IF in1 >= in2 AND in1 >= in3 THEN
	max3 := in1;
ELSIF in2 >= in1 AND in2 >= in3 THEN
	max3 := in2;
ELSE
	max3 := in3;
END_IF;

END_FUNCTION

// POUs/String/MESSAGE_4R
FUNCTION_BLOCK MESSAGE_4R
VAR_INPUT
	M0 : STRING(STRING_LENGTH);
	M1 : STRING(STRING_LENGTH);
	M2 : STRING(STRING_LENGTH);
	M3 : STRING(STRING_LENGTH);
	MM : INT := 3;
	ENQ : BOOL := TRUE;
	CLK : BOOL := TRUE;
	T1 : TIME := T#3s;
END_VAR
VAR_OUTPUT
	MX : STRING(STRING_LENGTH);
	MN : INT;
	TR : BOOL;
END_VAR
VAR
	timer : TON;
	edge: BOOL;
END_VAR

(*
version 1.1	27. oct. 2008
programmer 	hugo
tested by	tobias

this function generates a rotation meassage with up to 4 strings.
on each rising edge of EN the next message in line will be displayed.
when EN stays high longer then one cycle, the next message will be displayed automatically after the time T1 is elapsed.
the output MX is the generated message and CX is a counter 0..3 signaling the current message displayed.
the displayed messages are 0 .. MM.

*)

(* check for rising edge on EN *)
TR := FALSE;
IF ENQ THEN
	IF (NOT edge AND clk) OR timer.q THEN
			MN := INC1(MN, MM);
			TR := TRUE;
			timer(in := FALSE);
			CASE MN OF
				0 : MX := M0;
				1 : MX := M1;
				2 : MX := M2;
				3 : MX := M3;
			END_CASE;
	END_IF;
	edge := clk;
	timer( in := CLK, pt := T1);
ELSE
	MX := '';
	MN := 0;
END_IF;




(* revision history
hm	8. oct. 2008	rev 1.0
	original version

hm	27. oct. 2008	rev 1.1
	changed _INC to INC1

*)

END_FUNCTION_BLOCK

// POUs/String/MESSAGE_8
FUNCTION_BLOCK MESSAGE_8
VAR_INPUT
	IN1 : BOOL;
	IN2 : BOOL;
	IN3 : BOOL;
	IN4 : BOOL;
	IN5 : BOOL;
	IN6 : BOOL;
	IN7 : BOOL;
	IN8 : BOOL;
END_VAR
VAR_INPUT CONSTANT
	S1 : STRING(STRING_LENGTH);
	S2 : STRING(STRING_LENGTH);
	S3 : STRING(STRING_LENGTH);
	S4 : STRING(STRING_LENGTH);
	S5 : STRING(STRING_LENGTH);
	S6 : STRING(STRING_LENGTH);
	S7 : STRING(STRING_LENGTH);
	S8 : STRING(STRING_LENGTH);
END_VAR
VAR_OUTPUT
	M : STRING(STRING_LENGTH);
END_VAR
VAR
END_VAR

(*
version 1.1	29. mar. 2008
programmer 	hugo
tested by	tobias

this function generates one out of 4 messages specified by S1 .. S8.
the selected message will be presented at the output M.
In1 has higher priority then In2 which has higher priority then IN3 and in8 has the lowest priority.
*)

(* check if an alarm is present if yes set the output M otherwise clear M *)
IF in1 THEN
	M := S1;
ELSIF in2 THEN
	M := S2;
ELSIF in3 THEN
	M := S3;
ELSIF in4 THEN
	M := S4;
ELSIF in5 THEN
	M := S5;
ELSIF in6 THEN
	M := S6;
ELSIF in7 THEN
	M := S7;
ELSIF in8 THEN
	M := S8;
ELSE
	M := '';
END_IF;

(* revision history
hm	26.12.2007		rev 1.0
	original version

hm	29. mar. 2008	rev 1.1
	changed STRING to STRING(STRING_LENGTH)
*)

END_FUNCTION_BLOCK

// POUs/Engineering/measurements/METER_STAT
FUNCTION_BLOCK METER_STAT
VAR_INPUT
	IN : REAL;
	DI : DATE;
	RST : BOOL;
END_VAR
VAR_OUTPUT RETAIN
	Last_Day : REAL;
	Current_Day : REAL;
	Last_Week : REAL;
	Current_Week : REAL;
	Last_Month : REAL;
	Current_Month : REAL;
	Last_Year : REAL;
	Current_Year : REAL;
END_VAR
VAR RETAIN
	Year_Start : REAL;
	Month_Start : REAL;
	Week_Start : REAL;
	Day_Start : REAL;
	last_run: DATE;
END_VAR

(*
	version 1.1	7. oct. 2008
	programmer 	oscat
	tested BY	oscat

METER_STAT runs statistics of a metered value, it calculates the current week, day, month and year consumption and stores the corresponding last day, week, month and year value.

*)

IF rst THEN
	Last_Day := 0;
	Current_Day := 0;
	Day_start := IN;
	Last_week := 0;
	Current_week := 0;
	Week_start := in;
	Last_month := 0;
	Current_month := 0;
	month_start := in;
	last_year := 0;
	current_year := 0;
	year_start := in;
ELSE
	Current_Day := IN - Day_Start;
	Current_Week := In - Week_Start;
	Current_Month := IN - Month_Start;
	Current_Year := IN - Year_Start;
END_IF;

IF YEAR_OF_DATE(DI) > YEAR_OF_DATE(last_run) THEN
	(* a new year has started *)
	last_year := current_year;
	current_year := 0;
	year_start := in;
	last_month := current_month;
	current_month := 0;
	month_start := in;
	last_day := current_day;
	current_day := 0;
	day_start := in;
ELSIF MONTH_OF_DATE(DI) > MONTH_OF_DATE(last_run) THEN
	(* a new month has started, january is alrerady done by year change *)
	last_month := current_month;
	current_month := 0;
	month_start := in;
	last_day := current_day;
	current_day := 0;
	day_start := in;
ELSIF day_of_year(di) > day_of_year(last_run) THEN
	(* day has chaged, first day of year and first day of month has already been taken care of *)
	last_day := current_day;
	current_day := 0;
	day_start := in;
END_IF;
IF DAY_OF_WEEK(DI) < DAY_OF_WEEK(last_run) THEN
	(* a new week has started *)
	last_week := current_week;
	current_week := 0;
	week_start := in;
END_IF;
last_run := di;

(* revision history
hm	16. sep. 2007	rev 1.0
	original version

hm	7. oct. 2008	rev 1.1
	changed function year_to_year_of_date
	changed function month to month_of_date
	changed function weekday to day_of_week

*)

END_FUNCTION_BLOCK

// POUs/Mathematical/MID3
FUNCTION MID3 : REAL
VAR_INPUT
	in1 : REAL;
	in2 : REAL;
	in3 : REAL;
END_VAR
VAR
END_VAR

(*
version 1.1	1 jan 2007
programmer 	hugo
tested by		tobias

returns the mid value of 3 real inputs.

*)

IF (in1 <= in2) AND (in1 >= in3) OR (in1 >= in2) AND (in1 <= in3) THEN
	mid3 := in1;
ELSIF (in2 <= in1) AND (in2 >= in3) OR (in2 >= in1) AND (in2 <= in3) THEN
	mid3 := in2;
ELSE
	mid3 := in3;
END_IF;

(*
hm	1.1.2007	rev 1.1
	rewrote the function for better performance

*)

END_FUNCTION

// POUs/Mathematical/MIN3
FUNCTION MIN3 : REAL
VAR_INPUT
	in1 : REAL;
	in2 : REAL;
	in3 : REAL;
END_VAR
VAR
END_VAR

(*
version 1.0	1 jan 2007
programmer 	hugo
tested by		tobias

this function returns the lowest of 3 real values

*)

IF in1 <= in2 AND in1 <= in3 THEN
	min3 := in1;
ELSIF in2 <= in1 AND in2 <= in3 THEN
	min3 := in2;
ELSE
	min3 := in3;
END_IF;

END_FUNCTION

// POUs/Time&Date/MINUTE_OF_DT
FUNCTION MINUTE_OF_DT : INT
VAR_INPUT
	XDT : DT;
END_VAR
VAR
END_VAR


(*
	version 1.0	6. jun. 2008
	programmer 	oscat
	tested BY	oscat

MINUTE_OF_DT returns the current minute (minute of the hour) of a DT variable

*)

MINUTE_OF_DT := DWORD_TO_INT(DT_TO_DWORD(XDT) MOD 3600)/60;


(* revision history
hm		6.9.2008	rev 1.0
	original version


*)

END_FUNCTION

// POUs/Time&Date/MINUTE_TO_TIME
FUNCTION MINUTE_TO_TIME : TIME
VAR_INPUT
	IN : REAL;
END_VAR
VAR
END_VAR

(*
version 1.2	24. feb. 2009
programmer 	hugo
tested by		oscat

converts an amount of minutes in real to time

*)

MINUTE_TO_TIME := DWORD_TO_TIME(REAL_TO_DWORD(IN * 60000.0));


(* revision history
hm	4. aug 2006	rev 1.0
	original version

hm	14. mar 2008	rev 1.1
	rounded the input after the last digit

hm	24. feb. 2009	rev 1.2
	changed input to IN

*)

END_FUNCTION

// POUs/String/MIRROR
FUNCTION MIRROR : STRING(STRING_LENGTH)
VAR_INPUT
	str : STRING(STRING_LENGTH);
END_VAR
VAR
	pi : POINTER TO ARRAY[1..255] OF BYTE;
	po : POINTER TO BYTE;
	lx: INT;
	i: INT;
END_VAR

(*
version 1.1	29. mar. 2008
programmer 	hugo
tested by	tobias

this function reverses an input string.

*)

pi := ADR(str);
po := ADR(mirror);
lx := LEN(str);
FOR i := lx TO 1 BY - 1 DO
	po^ := pi^[i];
	po := po + 1;
END_FOR;
(* close output string *)
po^:= 0;


(* revision histroy
hm	4. feb. 2008	rev 1.0
	original release

hm	29. mar. 2008	rev 1.1
	changed STRING to STRING(STRING_LENGTH)
*)

END_FUNCTION

// POUs/Engineering/signal processing/MIX
FUNCTION MIX : REAL
VAR_INPUT
	A, B : REAL;
	M : REAL;
END_VAR
VAR
END_VAR

(*
version 1.0	19 nov 2007
programmer 	hugo
tested by		tobias

MIX is an analog Mixer. The Output is (1-M)*A + M*B.

*)

MIX := (1-M)*A + M*B;

(* revision history
hm	19. Nov 2007		rev 1.0
	original version
*)

END_FUNCTION

// POUs/Time&Date/MONTH_BEGIN
FUNCTION MONTH_BEGIN : DATE
VAR_INPUT
	idate : DATE;
END_VAR
VAR
END_VAR

(*
version 1.0	15. jun. 2008
programmer 	hugo
tested by	oscat

returns the date for the first day of the current month in the current year.

*)

MONTH_BEGIN := DWORD_TO_DATE(DATE_TO_DWORD(idate) - INT_TO_DWORD(DAY_OF_MONTH(idate) - 1) * 86400);



(* revision history
hm	15. jun. 2008	rev 1.0
	original version	


*)

END_FUNCTION

// POUs/Time&Date/MONTH_END
FUNCTION MONTH_END : DATE
VAR_INPUT
	IDATE : DATE;
END_VAR
VAR
END_VAR

(*
version 1.1	7. oct. 2008
programmer 	hugo
tested by	oscat

returns the date for the last day of the current month in the current year.

*)

MONTH_END := DWORD_TO_DATE(DATE_TO_DWORD(SET_DATE(YEAR_OF_DATE(idate),MONTH_OF_DATE(idate)+1,1)) - 86400);



(* revision history
hm	15. jun. 2008	rev 1.0
	original version	

hm	7. oct. 2008	rev 1.1
	changed function year to year_of_date
	changed function month to month_of_date

*)

END_FUNCTION

// POUs/Engineering/conversion/MS_TO_BFT
FUNCTION MS_TO_BFT : INT
VAR_INPUT
	MS : REAL;
END_VAR
VAR
END_VAR

(*
version 1.0	12. jun 2008
programmer 	hugo
tested by	oscdat

this function converts wind speed from M/s to beaufort
*)

MS_TO_BFT := REAL_TO_INT(EXPT(MS * 1.196172, 0.666667));


(* revision history
hm	12. 6. 2008		rev 1.0
	original version

*)

END_FUNCTION

// POUs/Engineering/conversion/MS_TO_KMH
FUNCTION MS_TO_KMH : REAL
VAR_INPUT
	ms : REAL;
END_VAR
VAR
END_VAR

(*
version 1.0	4 Feb 2007
programmer 	hugo
tested by		tobias

this function converts velocities from Meters / Second to Kilometers / hour.

*)

MS_TO_KMH := ms * 3.6;

END_FUNCTION

// POUs/Mathematical/MUL_ADD
FUNCTION MUL_ADD : REAL
VAR_INPUT
	X : REAL;
	K : REAL;
	O : REAL;
END_VAR
VAR
END_VAR

(*
version 1.1	11 nov 2007
programmer 	hugo
tested by		tobias

this function multiplies an input X with K and adds Offset O to the result.

*)

MUL_ADD := X * K + O;

(* revision history
hm	28. feb 2007
	original version

hm	11.nov 2007		rev 1.1
	deleted preset values for K and O this makes no sense for a function

*)

END_FUNCTION

// POUs/Engineering/sensor/MULTI_IN
FUNCTION MULTI_IN : REAL
VAR_INPUT
	in_1 : REAL;
	in_2 : REAL;
	in_3 : REAL;
	default : REAL;
	in_min : REAL;
	in_max : REAL;
	mode : BYTE;
END_VAR
VAR
	count: INT;
	F1: BOOL;
	F2: BOOL;
	F3: BOOL;
END_VAR

(*

version 1.2	14. oct. 2008
programmer 	oscat
tested by	oscat

multi_in is a signal conditioning function which can be configured in 8 different ways.
it is used to read multiple sensors for the same value and protect the user from broken sensors or invalid data from sensors.

multi_in can be configured in different ways:
	mode = 0 means the the avg of the 3 inputs is used, this mode is the default mode.
	mode = 1 means in_1 is used.
	mode = 2 means in_2 is used.
	mode = 3 means in_3 is used.
	mode = 4 means default is used.
	mode = 5 means the lowest of the 3 external temperatures is used.
	mode = 6 means the higest externnal temperature is used.
	mode = 7 means the midlle input is used, if there are only two working, the lowest input is used.
	mode > 7 ,eans output is 0 at all times.
	in any config mode, an input higher then in_max or lower then in_min is ignored to prevent values from broken sensors or wires.
	if all inputs are higher then in_max or lower then in_min, a default value (default) is used.
*)

F1 :=  in_1 > in_min AND in_1 < in_max;
F2 :=  in_2 > in_min AND in_2 < in_max;
F3 :=  in_3 > in_min AND in_3 < in_max;

CASE mode OF
0:	count := 0;
	IF F1 THEN
		count := count + 1;
		MULTI_IN := in_1;
	ELSE
		MULTI_IN := 0;
	END_IF;
	IF F2 THEN
		count := count + 1;
		MULTI_IN := MULTI_IN + in_2;
	END_IF;
	IF F3 THEN
		count := count + 1;
		MULTI_IN := MULTI_IN + in_3;
	END_IF;
	IF count = 0 THEN
		MULTI_IN := default;
	ELSE
		MULTI_IN := MULTI_IN / count;
	END_IF;

1:	IF F1 THEN MULTI_IN := in_1; ELSE MULTI_IN := default; END_IF;

2:	IF F2 THEN MULTI_IN := in_2; ELSE MULTI_IN := default; END_IF;

3:	IF F3 THEN MULTI_IN := in_3; ELSE MULTI_IN := default; END_IF;

4:	MULTI_IN := default;

5:	IF F1 THEN MULTI_IN := in_1; ELSE MULTI_IN := in_max; END_IF;
	IF F2 AND in_2 < MULTI_IN THEN MULTI_IN := in_2; END_IF;
	IF F3 AND in_3 < MULTI_IN THEN MULTI_IN := in_3; END_IF;
	IF MULTI_IN = in_max THEN MULTI_IN := default; END_IF;

6:	IF F1 THEN MULTI_IN := in_1; ELSE MULTI_IN := in_min; END_IF;
	IF F2 AND in_2 > MULTI_IN THEN MULTI_IN := in_2; END_IF;
	IF F3 AND in_3 > MULTI_IN THEN MULTI_IN := in_3; END_IF;
	IF MULTI_IN = in_min THEN MULTI_IN := default; END_IF;

7:	IF F1 AND F2 AND F3 THEN MULTI_IN := MID3(in_1, in_2, in_3);
	ELSIF F1 AND F2 THEN MULTI_IN := MIN(in_1, in_2);
	ELSIF F1 AND F3 THEN MULTI_IN := MIN(in_1, in_3);
	ELSIF F2 AND F3 THEN MULTI_IN := MIN(in_2, in_3);
	ELSIF F1 THEN MULTI_IN := in_1;
	ELSIF F2 THEN MULTI_IN := in_2;
	ELSIF F3 THEN MULTI_IN := in_3;
	ELSE MULTI_IN := default;
	END_IF;

END_CASE;

(*
hm 1.1.2007			rev 1.1
	changed midr to mid3 function

hm	14. 10. 2008	rev 1.2
	corrected an error for in_3 overrange detection
	improved performance


*)

END_FUNCTION

// POUs/Logic/gate logic/MUX_2
FUNCTION MUX_2 : BOOL
VAR_INPUT
	D0: BOOL;
	D1: BOOL;
	A0: BOOL;
END_VAR
VAR
END_VAR

(*
	version 1.2	16. oct. 2008
	programmer 	hugo
	tested BY	oscat

	dual input multiplexer
	depending on the value of A0, D0 or D1 will be switched to the Output

	executioin TIME on wago 750-841 = 7us
*)

MUX_2 := SEL(A0, D0, D1);


(*
revision history:
hm	5.10.2006		rev 1.1
	changed to ST Langage for better portability.

hm	16. oct. 2008	rev 1.2
	improved performance

*)

END_FUNCTION

// POUs/Logic/gate logic/MUX_4
FUNCTION MUX_4 : BOOL
VAR_INPUT
	D0: BOOL;
	D1: BOOL;
	D2: BOOL;
	D3: BOOL;
	A0: BOOL;
	A1: BOOL;
END_VAR
VAR
END_VAR

(*
version 1.2	16. oct. 2008
programmer 	hugo
tested BY	oscat

quad input multiplexer
depending on the value of A0 and A1, one of the 4 inputs will be switched to the Output


*)

IF A1 THEN
	MUX_4 := SEL(A0, D2, D3);
ELSE
	MUX_4 := SEL(A0, D0, D1);
END_IF;


(*
revision history:
hm 	5.10.2006		rev 1.1
	rewritten to ST for better portability

hm	16. oct. 2008	rev 1.2
	improved performance

*)

END_FUNCTION

// POUs/Engineering/signal processing/MUX_R2
FUNCTION MUX_R2 : REAL
VAR_INPUT
	IN0 : REAL;
	IN1 : REAL;
	A : BOOL;
END_VAR
VAR
END_VAR

(*
version 1.1	16. oct. 2008
programmer 	oscat
tested by	oscat

MUX_R2 is an analog Multiplexer.
one of 2 real inputs are selected and put through to out.
The Adress input A selects between 2 Real inputs IN0 and IN1, A=0 > In0, A=1 > in1.

*)

MUX_R2 := SEL(A, IN0, IN1);


(* revision history
hm	19. jan. 2007	rev 1.0
	original version

hm	16. oct. 2008	rev 1.1
	improved performance


*)

END_FUNCTION

// POUs/Engineering/signal processing/MUX_R4
FUNCTION MUX_R4 : REAL
VAR_INPUT
	IN0 : REAL;
	IN1 : REAL;
	IN2 : REAL;
	IN3 : REAL;
	A0 : BOOL;
	A1 : BOOL;
END_VAR
VAR
END_VAR

(*
version 1.1	16. oct. 2008
programmer 	oscat
tested by	oscat

MUX_R4 is an analog Multiplexer.
one of 4 real inputs are selected and put through to out.
The Adress input A0 and A1 selects between the 4 Real inputs IN0.. IN1.

*)

IF A1 THEN
	MUX_R4 := SEL(A0, IN2, IN3);
ELSE
	MUX_R4 := SEL(A0, IN0, IN1);
END_IF;



(* revision history
hm	19. jan 2007	rev 1.0
	original version

hm	16. oct. 2008	rev 1.1
	improved performance
*)

END_FUNCTION

// POUs/Mathematical/NEGX
FUNCTION NEGX : REAL
VAR_INPUT
	X : REAL;
END_VAR
VAR
END_VAR


(*
version 1.0	26. oct. 2008
programmer 	hugo
tested by	tobias

This function returns -X

*)

NEGX := -X;




(* revision history
hm	26. oct. 2008	rev 1.0
	original version


*)

END_FUNCTION

// POUs/Engineering/signal processing/OFFSET2
FUNCTION OFFSET2 : REAL
VAR_INPUT
	X : REAL;
	O1, O2, O3, O4 : BOOL;
	D : BOOL;
END_VAR
VAR_INPUT CONSTANT
	Offset_1 : REAL;
	Offset_2 : REAL;
	Offset_3 : REAL;
	Offset_4 : REAL;
	default : REAL;
END_VAR

(*
version 1.0	12 jan 2007
programmer 	oscat
tested by		tobias

The Function offset adds offsets to an analog signal depending on digital inputs.
one offset can be added at the same time, if more then one input is true, the one with the highest number (o1 .. o4) will be used.
The input D will select a default value instead of X for input.

*)

IF D THEN OFFSET2 := default; ELSE OFFSET2 := X; END_IF;
IF O4 THEN OFFSET2 := OFFSET2 + offset_4;
ELSIF O3 THEN OFFSET2 := OFFSET2 + offset_3;
ELSIF O2 THEN OFFSET2 := OFFSET2 + offset_2;
ELSIF O1 THEN OFFSET2 := OFFSET2 + offset_1;
END_IF;

END_FUNCTION

// POUs/Engineering/conversion/OM_TO_F
FUNCTION OM_TO_F : REAL
VAR_INPUT
	OM : REAL;
END_VAR
VAR
END_VAR

(*
version 1.1	18. oct. 2008
programmer 	hugo
tested by		tobias

this function converts Omega F to frequency
F = OM / (2*PI)
*)

OM_TO_F := OM / math.PI2;


(* revision history
hm	22. jan. 2007	rev 1.0
	original version

hm	18. oct. 2008	rev 1.1
	using math constants

*)

END_FUNCTION

// POUs/Other/OSCAT_VERSION
FUNCTION OSCAT_VERSION : DWORD
VAR_INPUT
	IN : BOOL;
END_VAR
VAR
END_VAR


(*
version 1.1	16 dec 2007
programmer 	hugo
tested by		oscat

oscat_version returns the version number in dword format
132 is library version 1.32
if IN = true, the release date will be returned

*)

IF in THEN
	OSCAT_VERSION := DATE_TO_DWORD(D#2009-3-1);
ELSE
	OSCAT_VERSION := 304;
END_IF;

(* revision history
hm	6. oct 2006	rev 1.0
	original version

hm	16. dec 2007	rev 1.1
	added possibility to return date and version depending on IN.

*)

END_FUNCTION

// POUs/Engineering/automation/PARSET
FUNCTION_BLOCK PARSET
VAR_INPUT
	A0, A1 : BOOL;
END_VAR
VAR_INPUT CONSTANT
	X01, X02, X03, X04 : REAL;
	X11, X12, X13, X14 : REAL;
	X21, X22, X23, X24 : REAL;
	X31, X32, X33, X34 : REAL;
	TC : TIME;
END_VAR
VAR_OUTPUT
	P1, P2, P3, P4 : REAL;
END_VAR
VAR
	X : ARRAY[0..3,1..4] OF REAL;
	S1, S2, S3, S4 : REAL;
	tx, last : DWORD;
	start : BOOL;
	set : BYTE;
	init: BOOL;
END_VAR

(*
version 1.1	16. mar. 2008
programmer 	hugo
tested by		tobias

parset selects on of 4 parameter sets adressed by the inputs A0 and A1. if TC is specified, the change of the outputs
is ramped by the time tc
*)

(* read system_time *)
tx := T_PLC_MS();

(* init sequence *)
IF NOT init THEN
	set.0 := NOT A0;
	init := TRUE;
	X[0,1] := X01;
	X[0,2] := X02;
	X[0,3] := X03;
	X[0,4] := X04;
	X[1,1] := X11;
	X[1,2] := X12;
	X[1,3] := X13;
	X[1,4] := X14;
	X[2,1] := X21;
	X[2,2] := X22;
	X[2,3] := X23;
	X[2,4] := X24;
	X[3,1] := X31;
	X[3,2] := X32;
	X[3,3] := X33;
	X[3,4] := X34;
	P1 := X01;
	P2 := X02;
	P3 := X03;
	P4 := X04;
END_IF;

(* check for input change *)
IF (A0 XOR set.0) OR (A1 XOR set.1) THEN
	(* a new set is selected *)
	set.0 := A0;
	set.1 := A1;
	IF tc > t#0s THEN
		start := TRUE;
		last := tx;
		(* save the step speed for the output changes in S *)
		S1 := (X[set,1] - P1)/DWORD_TO_REAL(TIME_TO_DWORD(tc));
		S2 := (X[set,2] - P2)/DWORD_TO_REAL(TIME_TO_DWORD(tc));
		S3 := (X[set,3] - P3)/DWORD_TO_REAL(TIME_TO_DWORD(tc));
		S4 := (X[set,4] - P4)/DWORD_TO_REAL(TIME_TO_DWORD(tc));
	END_IF;
ELSIF start AND tx - last < TIME_TO_DWORD(tc) THEN
	(* ramp the outputs to the new value *)
	P1 := X[set,1] - S1 * DWORD_TO_REAL(TIME_TO_DWORD(Tc) - tx + last);
	P2 := X[set,2] - S2 * DWORD_TO_REAL(TIME_TO_DWORD(Tc) - tx + last);
	P3 := X[set,3] - S3 * DWORD_TO_REAL(TIME_TO_DWORD(Tc) - tx + last);
	P4 := X[set,4] - S4 * DWORD_TO_REAL(TIME_TO_DWORD(Tc) - tx + last);
ELSE
	(* make sure outputs match the correct set values *)
	start := FALSE;
	P1 := X[set,1];
	P2 := X[set,2];
	P3 := X[set,3];
	P4 := X[set,4];
END_IF;

(* revision history
hm	2.11.2007		rev 1.0
	original version

hm	16. mar. 2008	rev 1.1
	added type conversions to avoid warnings under codesys 3.0

*)

END_FUNCTION_BLOCK

// POUs/Engineering/automation/PARSET2
FUNCTION_BLOCK PARSET2
VAR_INPUT
	X : REAL;
END_VAR
VAR_INPUT CONSTANT
	X01, X02, X03, X04 : REAL;
	X11, X12, X13, X14 : REAL;
	X21, X22, X23, X24 : REAL;
	X31, X32, X33, X34 : REAL;
	L1, L2, L3 : REAL;
	TC : TIME;
END_VAR
VAR_OUTPUT
	P1,P2,P3,P4 : REAL;
END_VAR
VAR
	Pset : parset;
	init: BOOL;
END_VAR

(*
version 1.0	3 nov 2007
programmer 	hugo
tested by	tobias

parset2 selects on of 4 parameter sets depending on the value of X. if TC is specified, the change of the outputs
is ramped by the time TC
*)

(* init sequence *)
IF NOT init THEN
	init := TRUE;
	pset(TC:=TC, X01:=X01, X02:=X02, X03:=X03, X04:=X04, X11:=X11, X12:=X12, X13:=X13, X14:=X14, X21:=X21, X22:=X22, X23:=X23, X24:=X24, X31:=X31, X32:=X32, X33:=X33, X34:=X34);
END_IF;
IF ABS(X) < L1 THEN
	pset(A0 := FALSE, A1 := FALSE);
ELSIF ABS(X) < L2 THEN
	pset(A0 := TRUE, A1 := FALSE);
ELSIF ABS(x) < L3 THEN
	pset(A0 := FALSE, A1 := TRUE);
ELSE
	pset(A0 := TRUE, A1 := TRUE);
END_IF;
P1 := pset.P1;
P2 := pset.P2;
P3 := pset.P3;
P4 := pset.P4;

(* revision history
hm		3.11.2007		rev 1.0
	original version

*)

END_FUNCTION_BLOCK

// POUs/Time&Date/PERIOD2
FUNCTION PERIOD2 : BOOL
VAR_INPUT
	DP : ARRAY[0..3,0..1] OF DATE;
	DX : DATE;
END_VAR
VAR
END_VAR

(*
version 1.0	27. apr. 2008
programmer 	hugo
tested by	tobias

PERIOD2 checks if DX is within one of 4 periods and sets the output true if so.

*)

PERIOD2 := 	(DX >= DP[0,0] AND DX <= DP[0,1]) OR
			(DX >= DP[1,0] AND DX <= DP[1,1]) OR
			(DX >= DP[2,0] AND DX <= DP[2,1]) OR
			(DX >= DP[3,0] AND DX <= DP[3,1]);


(* revision history

hm		27. apr 2008	rev 1.0
	original version


*)

END_FUNCTION

// POUs/Logic/Others/PIN_CODE
FUNCTION_BLOCK PIN_CODE
VAR_INPUT
	CB : BYTE;
	E : BOOL;
END_VAR
VAR_INPUT CONSTANT
	PIN : STRING(8);
END_VAR
VAR_OUTPUT
	TP : BOOL;
END_VAR
VAR
	POS: INT := 1;
END_VAR

(*
version 1.0	30. oct. 2008
programmer 	hugo
tested by	oscat

MATRIX_CODE scans the input of a key_pad (MATRIX) for a sequence of characters.

*)

tp := FALSE;
IF e THEN
	IF CB = CODE(pin, pos) THEN
		pos := pos + 1;
		IF pos > LEN(PIN) THEN
			(* proper code is detected *)
			TP := TRUE;
			pos := 1;
		END_IF;
	ELSE
		pos := 1;
	END_IF;
END_IF;


(* revision history
hm	30. oct. 2008	rev 1.0		
	original version 


*)

END_FUNCTION_BLOCK

// POUs/Mathematical/functions/POLYNOM_INT
FUNCTION POLYNOM_INT : REAL
VAR_INPUT
	X : REAL;
	XY : ARRAY[1..5,0..1] OF REAL;
	Pts : INT;
END_VAR
VAR
	I, J : INT;
	stop: INT;
END_VAR

(*
	version 1.2	22 feb 2008
	programmer 	oscat
	tested BY		oscat

POLYNOM_INT calculates an output based on a Polynom interpolation of up to 5 coordinates given in an array
the indut coordinates have to start at the lowest array position and must be sorted ba ascending X values.

*)

(*make sure n is bound within the array size *)
pts := MIN(pts, 5);

(* this part is only to calculate the polynom parameters, which are then stores in the Y array
	the array values, it is not needed during runtime, unless the parameters will change during runtime
	the remaining code without this setup code can be used within a function to calculate specific functions
	the content of the arrays is then used as constant values within the function *)

FOR i := 1 TO pts DO
	stop := i + 1;
   	FOR j := pts TO stop BY -1 DO
   		XY[j,1] := (XY[j,1] - XY[j-1,1]) / (XY[j,0] - XY[j-i,0]);
	END_FOR;
END_FOR;


(* this part is the actual calculation *)
POLYNOM_INT := 0;
FOR i := pts TO 1 BY -1 DO
       POLYNOM_INT := POLYNOM_INT * (X - XY[i,0]) + XY[i,1];
END_FOR;


(* revision history
hm		8. okt 2007		rev 1.0
	original version

hm		17. dec 2007	rev 1.1
	init makes no sense for a function

hm		22. feb 2008	rev 1.2
	improved performance
*)

END_FUNCTION

// POUs/Engineering/conversion/PT_TO_F
FUNCTION PT_TO_F : REAL
VAR_INPUT
	PT : TIME;
END_VAR
VAR
END_VAR

(*
version 1.0	4 aug 2006
programmer 	hugo
tested by		tobias

this function converts periode time to frequency
*)

PT_to_F := 1000/DWORD_TO_REAL(TIME_TO_DWORD(PT));

END_FUNCTION

// POUs/Building/electrical/PULSE_LENGTH
FUNCTION_BLOCK PULSE_LENGTH
VAR_INPUT
	in : BOOL;
END_VAR
VAR_OUTPUT
	short : BOOL;
	middle : BOOL;
	long : BOOL;
END_VAR
VAR_INPUT CONSTANT
	T_short : TIME := t#100ms;
	T_long : TIME := t#1s;
END_VAR
VAR
	tx : TIME;
	tn: TIME;
	edge : BOOL;
END_VAR

(*
version 1.1	15 sep 2007
programmer 	oscat
tested by	oscat

Pulse_length indicates on 3 outputs if an input pulse had been shorter than T_short (short = True), longer than T_long (long = True) or between T_short and T_long (middle = True).

*)

(* read system time *)
tx := DWORD_TO_TIME(T_PLC_MS());

(* reset outputs, they should only be active 1 cycle *)
short := FALSE;
Middle := FALSE;
long := FALSE;

(* detect rising edge *)
IF in AND NOT edge THEN
	edge := TRUE;
	tn := tx;

(* detect for falling edge *)
ELSIF NOT in AND edge THEN
	edge := FALSE;
	tn := tx - tn;
	IF tn < t_short THEN
		short := TRUE;
	ELSIF tn > t_long THEN
		long := TRUE;
	ELSE
		Middle := TRUE;
	END_IF;

(* generate long pulse as soon as T_long is reached *)
ELSIF in AND tx - tn > t_long THEN
	long := TRUE;
END_IF;


(* revision history

hm	15. feb 2006	rev 1.0
	original version

hm	15 sep 2007		rev 1.1
	replaced Time() with T_PLC_MS for compatibility and performance reasons

*)

END_FUNCTION_BLOCK

// POUs/Building/electrical/PULSE_T
FUNCTION_BLOCK PULSE_T
VAR_INPUT
	IN : BOOL;
	T1 : TIME;
	T2 : TIME;
	RST : BOOL;
END_VAR
VAR_OUTPUT
	Q : BOOL;
END_VAR
VAR
	init: BOOL;
	last: TIME;
	tx: TIME;
	edge: BOOL;
END_VAR


(*
version 1.0	15. jul. 2008
programmer 	hugo
tested by	oscat

PULSE_T generates a pulse of length T2 if the input pulse is shorter than T1.
if the input pulse is longer than T1, the output follows the input.
and rising edge on in will kill a possible output pulse and generate a new pulse instead.

*)

tx := DWORD_TO_TIME(T_PLC_MS());
IF NOT init THEN
	init := TRUE;
	last := tx;
ELSIF RST THEN
	(* asynchronous reset *)
	Q := FALSE;
ELSIF IN AND NOT edge AND NOT Q THEN
	(* a rising edge on in will reversre the output status, if new pulse is startet the start time is stored in last *)
	last := tx;
	Q := TRUE;
ELSIF NOT IN AND edge AND ((tx - last) > T1) THEN
	(* a falling edge on IN will clear the output if in was high for more then T1 *)
	Q := FALSE;
ELSIF (tx - last) >= T2 THEN
	(* timeout for long pulse if second click did not occur or in stays high *)
	Q := FALSE;
END_IF;

edge := IN;

(* revision histroy
hm	15. jul. 2008	rev 1.0
	original release


*)

END_FUNCTION_BLOCK

// POUs/Engineering/signal generators/PWM_PW
FUNCTION_BLOCK PWM_PW
VAR_INPUT
	F : REAL;
	PW : TIME;
END_VAR
VAR_OUTPUT
	Q : BOOL;
END_VAR
VAR
	clk: CLK_PRG;
	pulse: TP_X;
END_VAR

(*
version 1.4	19. oct. 2008
programmer 	oscat
tested BY	oscat

this signal generator generates a square wave signal which is specified by the frequency and the pulse width.
*)

IF F > 0 THEN
	CLK(PT := REAL_TO_TIME(1000/F));
	Pulse(in := clk.Q, pt := pw);
	Q := pulse.Q;
END_IF;

(* revision history

hm	25. feb 2007	rev 1.1
	recoded in st for better performance and better portability

hm	27. nov 2007	rev 1.2
	avoid divide by 0 when F = 0

hm	9. dec 2007		rev 1.3
	corrected an error with F = 0

hm	19. oct. 2008	rev 1.4
	changed type tp_r to TP_x brecause of name change

*)

END_FUNCTION_BLOCK

// POUs/Mathematical/Double Precision/R2_ABS
FUNCTION R2_ABS : REAL2
VAR_INPUT
	X : REAL2;
END_VAR
VAR
END_VAR

(*
version 1.0	21. mar. 2008
programmer 	hugo
tested by		tobias

R2_abs returns the absulute value of a double precision real.

*)

IF X.RX >= 0 THEN
	R2_ABS.RX := X.RX;
	R2_ABS.R1 := X.R1;
ELSE
	R2_ABS.RX := ABS(X.RX);
	R2_ABS.R1 := -X.R1;
END_IF;


(* revision history
hm	21. mar. 2008	rev 1.0
	original version

*)

END_FUNCTION

// POUs/Mathematical/Double Precision/R2_ADD2
FUNCTION R2_ADD2 : REAL2
VAR_INPUT
	X : Real2;
	Y : REAL2;
END_VAR
VAR
END_VAR

(*
version 1.0	20. mar. 2008
programmer 	hugo
tested by		tobias

R2_add2 adds a double precision real to a double precision real which extends the accuracy of a real to twice as many digits

*)

R2_ADD2.R1 := X.R1 + Y.R1;
R2_ADD2.RX := X.RX + Y.RX;


(* revision history
hm		20.3.2008	rev 1.0
	original version

*)

END_FUNCTION

// POUs/Mathematical/Double Precision/R2_MUL
FUNCTION R2_MUL : REAL2
VAR_INPUT
	X : REAL2;
	Y : REAL;
END_VAR
VAR
END_VAR

(*
version 1.0	20. mar. 2008
programmer 	hugo
tested by		tobias

R2_mul multiplies a real with a double real which extends the accuracy of a real to twice as many digits

*)

R2_MUL.RX := X.RX * Y;
R2_MUL.R1 := X.R1 * Y;


(* revision history
hm		20.3.2008	rev 1.0
	original version

*)

END_FUNCTION

// POUs/Engineering/signal processing/RANGE_TO_BYTE
FUNCTION RANGE_TO_BYTE : BYTE
VAR_INPUT
	X : REAL;
	low : REAL;
	high : REAL;
END_VAR
VAR
END_VAR

(*
version 1.0	9. jan 2008
programmer 	hugo
tested by		tobias

Range_to_byte converts a real value between low and high into a byte

*)

Range_to_Byte := INT_TO_BYTE(TRUNC_INT((LIMIT(low,X,high)-low) * 255.0 / (high - low)));


(* revision history
hm	9. jan 2008		rev 1.0
	original version

*)

END_FUNCTION

// POUs/Engineering/signal processing/RANGE_TO_WORD
FUNCTION RANGE_TO_WORD : WORD
VAR_INPUT
	X : REAL;
	low : REAL;
	high : REAL;
END_VAR
VAR
END_VAR

(*
version 1.0	9. jan 2008
programmer 	hugo
tested by		tobias

Range_to_word converts a real value between low and high into a byte

*)

Range_to_Word := DINT_TO_WORD(TRUNC_INT((LIMIT(low,X,high)-low) * 65535.0 / (high - low)));


(* revision history
hm	9. jan 2008		rev 1.0
	original version

*)

END_FUNCTION

// POUs/Mathematical/RDMDW
FUNCTION RDMDW : DWORD
VAR_INPUT
	last : DWORD;
END_VAR
VAR
	RX: REAL;
	M: REAL;
END_VAR




(*
version 1.2	18. oct. 2008
programmer 	hugo
tested by		tobias

this function calculates a DWORD pseudo random number.

*)

M := BIT_COUNT(last);
RX := RDM(FRACT(M * math.PI));
RDMDW := SHL(REAL_TO_DWORD(rx*65535),16);
RX := RDM(FRACT(M * math.E));
RDMDW := RDMDW OR (REAL_TO_DWORD(rx*65535) AND 16#0000FFFF);



(* revision history
hm		14. mar 2008		rev 1.0
	original version

hm		18. may. 2008		rev 1.1
	changed constant E to E1

hm		18. oct. 2008		rev 1.2
	using math constants

*)

END_FUNCTION

// POUs/String/REAL_TO_STRF
FUNCTION REAL_TO_STRF : STRING(20)
VAR_INPUT
	IN : REAL;
	N : INT;
END_VAR
VAR
	O: REAL;
	i: INT;
END_VAR

(*
version 1.7	27. feb. 2009
programmer 	hugo
tested by		oscat

Real_to_strF converts a Real to a fixed length String.
the string will be filles with zeroes to achieve the fixed length after the dot.


*)

(* LIMIT N to 0 .. 7 *)
N := LIMIT(0,N,7);
(* round the input to N digits and convert to string *)
O := ABS(in) * EXP10(N);
REAL_TO_STRF := DINT_TO_STRING(REAL_TO_DINT(O));
(* add zeroes in front to make sure sting is at least 8 digits long *)
FOR i := LEN(REAL_TO_STRF) TO N DO REAL_TO_STRF := CONCAT('0', REAL_TO_STRF); END_FOR;
(* add a dot if n > 0 *)
IF n > 0 THEN REAL_TO_STRF := INSERT(REAL_TO_STRF, '.', LEN(REAL_TO_STRF) - N); END_IF;
(* add a minus sign if in is negative *)
IF in < 0 THEN REAL_TO_STRF := CONCAT('-', REAL_TO_STRF); END_IF;


(* revision history
hm	26 jan 2007	rev 1.0
	original version

hm	20. nov. 2007	rev 1.1
	when N=0 ther will be no dot at the end of the string.

hm	15. dec. 2007	rev 1.2
	changed code for better performance

hm	4. mar. 2008	rev 1.3
	result is now rounded instead of trunc

hm	20. mar. 2008	rev 1.4
	changed trunc to real_to_dint because trunc was generating wrong values on wago 842

hm	29. mar. 2008	rev 1.5
	changed STRING to STRING(20)

hm	4. apr. 2008	rev 1.6
	added variable O to avoid an error uner CoDeSys SP PLCWinNT V2.4

hm	27. feb. 2009	rev 1.7
	added a missing zero for IN < 1

*)

END_FUNCTION

// POUs/Mathematical/ROUND
 FUNCTION ROUND : REAL
VAR_INPUT
	in : REAL;
	N : INT;
END_VAR
VAR
	X: REAL;
END_VAR


(*
version 1.5	25. oct. 2008
programmer 	hugo
tested by	tobias

this function rounds a real down to n digits behind the comma.


*)

x := setup.DECADES[LIMIT(0,n,8)];
ROUND := DINT_TO_REAL(REAL_TO_DINT(in * X)) / X;



(* revision history
hm	1. sep 2006	rev 1.0
	original version

hm	2. dec 2007	rev 1.1
	changed code for better performance

hm	8. jan 2008	rev 1.2
	further improvement in performance

hm 11. mar. 2008	rev 1.3
	corrected an error with negative numbers
	use real_to_dint instead of trunc

hm	16. mar 2008	rev 1.4
	added type conversion to avoid warning under codesys 3.0

hm	25. oct. 2008	rev 1.5
	new code using global constants decades
*)

END_FUNCTION

// POUs/String/REPLACE_ALL
FUNCTION REPLACE_ALL : STRING(STRING_LENGTH)
VAR_INPUT
	str : STRING(STRING_LENGTH);
	src : STRING(STRING_LENGTH);
	rep : STRING(STRING_LENGTH);
END_VAR
VAR
	pos: INT;
	lp : INT;
	lx : INT;
END_VAR

(*
version 1.1	29. mar. 2008
programmer 	hugo
tested by	tobias

the function replace_all replaces all occurences of src in str and replaces them by rep.

*)

REPLACE_ALL := str;
lx := LEN(src);
lp := LEN(rep);
pos := FINDP(REPLACE_ALL, src, 1);
WHILE pos > 0 DO
	REPLACE_ALL := REPLACE(REPLACE_ALL,rep,lx, pos);
	pos := FINDP(REPLACE_ALL, src, pos + lp);
END_WHILE;

(* revision histroy
hm	4. feb. 2008	rev 1.0
	original release

hm	29. mar. 2008	rev 1.1
	changed STRING to STRING(STRING_LENGTH)
*)

END_FUNCTION

// POUs/String/REPLACE_CHARS
FUNCTION REPLACE_CHARS : STRING(STRING_LENGTH)
VAR_INPUT
	STR : STRING(STRING_LENGTH);
	SRC : STRING;
	REP : STRING;
END_VAR
VAR
	a, b : INT;
	c: STRING(1);
	stp: INT;
END_VAR

(*
version 1.0		14. may. 2008
programmer 		hugo
tested by			hugo

REPLACE_CHARS erstezt alle character die im string src aufgeführt sind mit dem an der selben stelle im string rep gelisteten character.

*)

REPLACE_CHARS := STR;
(* make sure rep and src are of same length and length is > 0 *)
a := LEN(src);
b := LEN(rep);
IF a < b THEN
	rep := LEFT(rep, a);
ELSIF b < a THEN
	src := LEFT(src, b);
END_IF;

(* search the string and replace if necessary *)
stp := LEN(str);
FOR a := 1 TO stp DO
	c := MID(REPLACE_CHARS, 1, a);
	b := FIND(src, c);
	IF b > 0 THEN
		REPLACE_CHARS := REPLACE(REPLACE_CHARS, MID(rep, 1, b), 1, a);
	END_IF;
END_FOR;



(* revision history
hm	14. may. 2008	rev 1.0
	original version

*)

END_FUNCTION

// POUs/String/REPLACE_UML
FUNCTION REPLACE_UML : STRING(STRING_LENGTH)
VAR_INPUT
	str : STRING(STRING_LENGTH);
END_VAR
VAR
	L : INT;
	pt : POINTER TO BYTE;
	pto : POINTER TO BYTE;
	ptm : POINTER TO BYTE;
	pt1, pt2 : POINTER TO BYTE;
	su : STRING(2);
	pos : INT;
END_VAR

(*
version 1.1	29. mar. 2008
programmer 		kurt
tested by		hugo

REPLACE_UML replaces all occurences of Ä,Ö,Ü and ä,ö,ü,ß with Ae, ae, Oe, oe, Ue, ue and ss.

*)

PT := ADR(str);
pto := ADR(REPLACE_UML);
ptm := pto + INT_TO_DWORD(string_length);
pt1 := ADR(su);
pt2 := pt1 + 1;
L := LEN(str);
WHILE pos < L AND pos < string_length DO
	IF pt^ < 127 THEN
		(* no uml character simlply copy the character*)
		pto^ := pt^;
	ELSE
		(* convert the uml character *)
		su := TO_UML(pt^);
		(* we must make sure pointer are not out of range *)
		pto^ := pt1^;
		IF pto < ptm AND pt2^ > 0 THEN
			pto := pto + 1;
			pto^ := pt2^;
		END_IF;
	END_IF;
	(* increment pointers *)
	pt := pt + 1;
	pto := pto + 1;
	pos := pos + 1;
END_WHILE;

(* properly close the output string *)
pto^ := 0;


(* revision history
hm	29. feb 2008	rev 1.0
	original version

hm	29. mar. 2008	rev 1.1
	changed STRING to STRING(STRING_LENGTH)
	new code to avoid pointer out of range
	use new function to_uml
*)

END_FUNCTION

// POUs/String/TO_UML
FUNCTION TO_UML : STRING(2)
VAR_INPUT
	IN : BYTE;
END_VAR
VAR
END_VAR

(*
version 1.1	17. dec. 2008
programmer 		hugo
tested by		tobias

to_uml converts a character above 127 to a two digit character below 127.
the character Ä is converted to Ae

*)

CASE in OF
	196:	(* Ä *)
		TO_UML := 'Ae';
	214:	(* Ö *)
		TO_UML := 'Oe';
	220:	(* Ü *)
		TO_UML := 'Ue';
	223:	(* ß *)
		TO_UML := 'ss';
	228:	(* ä *)
		TO_UML := 'ae';
	246:	(* ö *)
		TO_UML := 'oe';
	252:	(* ü *)
		TO_UML := 'ue';
ELSE
	TO_UML := CHR_TO_STRING(IN);
END_CASE;



(* revision history
hm	29. mar. 2008	rev 1.0
	original version

hm	17. dec. 2008	rev 1.1
	changes name of function chr to chr_to_string

*)

END_FUNCTION

// POUs/Engineering/sensor/RES_NI
FUNCTION RES_NI : REAL
VAR_INPUT
	T : REAL;
	R0 : REAL;
END_VAR
VAR CONSTANT
	A : REAL := 0.5485;
	B : REAL := 0.665E-3;
	C : REAL := 2.805E-9;
END_VAR
VAR
	T2: REAL;
END_VAR

(*
version 1.2	2 dec 2007
programmer 	hugo
tested by		tobias

this function returs the resistance for a nickel sensor for a temperature range from -60..+180 °C *)

T2 := T*T;
Res_NI := R0 + A*T + B*T2 + C*T2*T2;

(* revision history

hm	4.8.2006		rev 1.0
	original version

hm	13.9.2007		rev 1.1
	changed coding for better performance

hm	2. dec. 2007	rev 1.2
	changed code for better performance
*)

(*

 Auszug aus DIN 43760 für Ni100

°C		R		°C		R		°C	R		°C		R		°C		R

-60 	69,5 	-10 	94,6 	40 	123,0 	90 		154,9 	140 	190,9
-55 	71,9 	-5 		97,3 	45 	126,0 	95 		158,3 	145 	194,8
-50 	74,3 	0 		100,0 	50 	129,1 	100 	161,8 	150 	198,7
-45 	76,7 	5 		102,8 	55 	132,2 	105 	165,3 	155 	202,6
-40 	79,1 	10 		105,6 	60 	135,3 	110 	168,8 	160 	206,6
-35 	81,6 	15 		108,4 	65 	138,5 	115 	172,4 	165 	210,7
-30 	84,2 	20 		111,2 	70 	141,7 	120 	176,0 	170 	214,8
-25 	86,7 	25 		114,1 	75 	145,0 	125 	179,6 	175 	219,0
-20 	89,3 	30 		117,1 	80 	148,3 	130 	183,3 	180 	223,2
-15 	91,9 	35 		120,0 	85 	151,6 	135 	187,1 	  	 

*)

END_FUNCTION

// POUs/Engineering/sensor/RES_NTC
FUNCTION RES_NTC : REAL
VAR_INPUT
	T : REAL;
	RN : REAL;
	B : REAL;
END_VAR


(*
version 1.0	30. dec. 2008
programmer 	hugo
tested by		tobias

this function returs the resistance for a NTC sensor for a given temperature in °C.
RN is the resistance at 25 °C and B is a constant for the given sensor.

*)

RES_NTC := RN * EXP(B * (1/(T+273.15) - 0.00335401643468053));



(* revision history

hm 30. dec. 2008	rev 1.0
	original version


*)

END_FUNCTION

// POUs/Engineering/sensor/RES_PT
FUNCTION RES_PT : REAL
VAR_INPUT
	T : REAL;
	R0 : REAL;
END_VAR
VAR CONSTANT
	A : REAL := 3.90802E-3 ;
	B : REAL := -5.802E-7;
	C : REAL := -4.27350E-12;
END_VAR
VAR
	T2: REAL;
END_VAR

(*
version 1.2	2. dec. 2007
programmer 	hugo
tested by	oscat


this function returs the resistance for a platinum sensor for a temperature range from -200..+850 °C *)

T2 := T * T;

IF T >= 0 THEN
	RES_PT := R0 * ( 1 + A*T + B*T2);
ELSE
	RES_PT := R0 * ( 1 + A*T + B*T2 + C*(T-100)*T2*T);
END_IF;



(* revision history
hm	4. aug. 2006	rev 1.1
	original version

hm	2. dec 2007		rev 1.2
	changed code for better performance


*)


(*
 Auszug aus DIN 43760 für Pt100

°C		R		°C		R		°C	R			°C		R			°C		R			°C		R

-200 	18,49 	-100 	60,25 	0 	100,00 	100 	138,50 	200 	175,84 	300 	212,02
-195 	20,65 	-95 	62,28 	5 	101,95 	105 	140,39 	205 	177,68 	305 	213,80
-190 	22,80 	-90 	64,30 	10 	103,90 	110 	142,29 	210 	179,51 	310 	215,57
-185 	24,94 	-85 	66,31 	15 	105,85 	115 	144,17 	215 	181,34 	315 	217,35
-180 	27,08 	-80 	68,33 	20 	107,79 	120 	146,06 	220 	183,17 	320 	219,12
-175 	29,20 	-75 	70,33 	25 	109,73 	125 	147,94 	225 	184,99 	325 	220,88
-170 	31,32 	-70 	72,33 	30 	111,67 	130 	149,82 	230 	186,82 	330 	222,65
-165 	33,43 	-65 	74,33 	35 	113,61 	135 	151,70 	235 	188,63 	335 	224,41
-160 	35,33 	-60 	76,33 	40 	115,54 	140 	153,58 	240 	190,45 	340 	226,17
-155 	37,63 	-55 	78,32 	45 	117,47 	145 	155,45 	245 	192,26 	345 	227,92
-150 	39,71 	-50 	80,31 	50 	119,40 	150 	157,31 	250 	194,07 	350 	229,67
-145 	41,79 	-45 	82,29 	55 	121,32 	155 	159,18 	255 	195,88 	355 	231,42
-140 	43,87 	-40 	84,27 	60 	123,24 	160 	161,04 	260 	197,69 	360 	233,17
-135 	45,94 	-35 	86,25 	65 	125,16 	165 	162,90 	265 	199,49 	365 	234,91
-130 	48,00 	-30 	88,22 	70 	127,07 	170 	164,76 	270 	201,29 	370 	236,65
-125 	50,06 	-25 	90,19 	75 	128,98 	175 	166,61 	275 	203,08 	375 	238,39
-120 	52,11 	-20 	92,16 	80 	130,89 	180 	168,46 	280 	204,88 	380 	240,13
-115 	54,15 	-15 	94,12 	85 	132,80 	185 	170,31 	285 	206,67 	385 	241,86
-110 	56,19 	-10 	96,09 	90 	134,70 	190 	172,16 	290 	208,45 	390 	243,59
-105 	58,22 	-5 		98,04 	95 	136,60 	195 	174,00 	295 	210,24 	395 	245,31

*)
(*
revision history


*)

END_FUNCTION

// POUs/Engineering/sensor/RES_SI
FUNCTION RES_SI : REAL
VAR_INPUT
	T : REAL;
	RS : REAL;
	TS : REAL;
END_VAR
VAR CONSTANT
	A : REAL := 7.64E-3;
	B : REAL := 1.66E-5;
END_VAR
VAR
	TX: REAL;
END_VAR

(*
version 1.1	2 dec 2007
programmer 	hugo
tested by		tobias

this function returs the resistance for a silicon sensor for a temperature range from -50..+150 °C
for example KTY10 normaly Rs at 25 °C
*)

TX := T - TS;
RES_SI := RS * ( 1 + A * TX + B * TX * TX);

(* revision history
hm		4. aug 2006		rev 1.0
	original version

hm		2. dec 2007		rev 1.1
	changed code for better performance

*)

END_FUNCTION

// POUs/Engineering/signal generators/RMP_SOFT
FUNCTION_BLOCK RMP_SOFT
VAR_INPUT
	IN : BOOL;
	VAL : BYTE;
END_VAR
VAR_INPUT CONSTANT
	PT_ON: TIME;
	PT_OFF : TIME;
END_VAR
VAR_OUTPUT
	OUT : BYTE;
END_VAR
VAR
	rmp : _RMP_B;
	tmp: BYTE;
END_VAR

(*
version 2.0	26. oct. 2008
programmer 	oscat
tested BY		oscat

this soft on/off ramp generator generates a soft on and soft off ramp while the max on value is set by the input
the time for a full ramp can be set by config variables for up and down ramp.

*)

tmp := SEL(in, 0, val);
IF tmp > out THEN
	(* we need to ramp down *)
	rmp(dir := TRUE, E := TRUE, TR := PT_ON, rmp := out);
	(* make sure out does not surpass tmp *)
	out := MIN(out, tmp);
ELSIF tmp < out THEN
	(* we need to ramp up *)
	rmp(dir := FALSE, E := TRUE, TR := PT_OFF, rmp := out);
	(* make sure out does not surpass tmp *)
	out := MAX(out, tmp);
ELSE
	(* no ramp necessary *)
	rmp(E := FALSE, rmp := out);
END_IF;


(* revision history

hm 22.1.2007	rev 1.1
	deleted unused variables X1 and I, X2 and X3

hm	17.9.2007	rev 1.2
	replaced time() with t_plc_ms() for compatibility reasons

hm	26. oct. 2008	2.0
	new code using _rmp_b
*)

END_FUNCTION_BLOCK

// POUs/Mathematical/RND
FUNCTION RND : REAL
VAR_INPUT
	X : REAL;
	N : INT;
END_VAR
VAR
	M : REAL;
END_VAR

(*
version 1.1	26. oct. 2008
programmer 	hugo
tested by	tobias

this function rounds a real down to n digits total.
round(3.1415,2) = 3.1

*)

IF X = 0 THEN
	RND := 0;
ELSE
	M := EXPN(10,N - CEIL(LOG(ABS(X))));
	RND := DINT_TO_REAL(REAL_TO_DINT(X * M)) / M;
END_IF;



(* revision history
hm	11. mar 2008	rev 1.0
	original version

hm	26. oct. 2008	rev 1.1
	code optimization
*)

END_FUNCTION

// POUs/Time&Date/RTC_2
FUNCTION_BLOCK RTC_2
VAR_INPUT
	SET : BOOL;
	SDT : DT;
	SMS : INT;
	DEN : BOOL;
	OFS : INT;
END_VAR
VAR_OUTPUT
	UDT : DT;
	LDT : DT;
	DSO : BOOL;
	XMS : INT;
END_VAR
VAR
	RT : RTC_MS;
END_VAR

(*
version 1.2	12. jun. 2008
programmer 	hugo
tested by	tobias

RTC_2 is a real time clock module which runs utc and generates local time from utc.
daylight savings time can be enabled with den and an additional local time is generated with a delay of ofs.

*)

(* call rtc *)
RT(SET := SET, SDT := SDT, SMS := SMS);
UDT := rt.xdt;
XMS := rt.XMS;

(* check for daylight savings time and set dso output *)
DSO := DST(udt) AND DEN;

(* calculate time offset and set ldt output *)
LDT := DWORD_TO_DT(DT_TO_DWORD(UDT) + INT_TO_DWORD(ofs + BOOL_TO_INT(DSO)) * 3600);


(* revision history
hm		20. jan. 2008	rev 1.0
	original version

hm		20. feb. 2008	rev 1.1
	added Millisecond Set input

hm		12. jun. 2008	rev 1.2
	improved performance
*)

END_FUNCTION_BLOCK

// POUs/Time&Date/RTC_MS
FUNCTION_BLOCK RTC_MS
VAR_INPUT
	SET : BOOL;
	SDT : DT;
	SMS : INT;
END_VAR
VAR_OUTPUT
	XDT : DT;
	XMS : INT;
END_VAR
VAR
	init: BOOL;
	last: DWORD;
	Tx: DWORD;
END_VAR

(*
version 1.1	20. feb. 2008
programmer 	hugo
tested by	tobias

RTC_MS is a real time clock module which can be set to SDT when set is TRUE and the outputs XDT and XT present the DateTime and TOD with a resolution of milliseconds.

*)

tx := T_PLC_MS();
IF set OR NOT init THEN
	(* clock needs to be set when set is true or after power up *)
	init := TRUE;
	xdt := SDT;
	XMS := SMS;
ELSE
	XMS := XMS + DWORD_TO_INT(tx - last);
	(* check if one second has expired *)
	IF XMS > 999 THEN
		XDT := XDT + T#1s;
		XMS := XMS - 1000;
	END_IF;
END_IF;
last := tx;


(* revision history
hm		20. jan. 2008	rev 1.0
	original version

hm		20. feb. 2008	rev 1.1
	added Millisecond Set input
*)

END_FUNCTION_BLOCK

// POUs/Engineering/signal processing/SCALE_B
FUNCTION SCALE_B : REAL
VAR_INPUT
	X : BYTE;
	I_LO : BYTE;
	I_HI : BYTE;
	O_LO : REAL;
	O_HI : REAL;
END_VAR
VAR
END_VAR

(*
version 1.0	18. may. 2008
programmer 	hugo
tested by		tobias

Scale_B is used to translate and scale a byte input x to a real output.

*)

SCALE_B := (O_HI - O_LO) / BYTE_TO_REAL(I_HI - I_LO) * BYTE_TO_REAL(LIMIT(I_LO,X,I_HI));


(* revision history
hm	18. may. 2008		rev 1.0
	original version
*)

END_FUNCTION

// POUs/Engineering/signal processing/SCALE_B2
FUNCTION SCALE_B2 : REAL
VAR_INPUT
	in1: BYTE;
	in2: BYTE;
	K : REAL;
	O : REAL;
END_VAR
VAR_INPUT CONSTANT
	in1_min: REAL;
	in1_max: REAL := 1000;
	in2_min: REAL;
	in2_max: REAL := 1000;
END_VAR

(*
version 1.4	3. nov. 2008
programmer 	hugo
tested by	oscat

this functiob block can scale up to two inputs.
inputs have their min value at 0 and their max value at 255 while the min and max value can be either positive or negative.
inputs ramp between min and max values for the respective inputs to be between (0..255).
the summed output is then scaled by an scale input K and a offset O can be added to the output.
min and max input configurations can be edited in the cfc editor by double clicking the symbol body.

*)

SCALE_B2 := 	(((in1_max - in1_min)* in1 + (in2_max - in2_min)* in2) * 0.003921569 + in1_min + in2_min) * K + O;

(* code bofore rev 1.2
scale_B2 := 	((in1_max - in1_min)* in1 / 255 + in1_min +
				(in2_max - in2_min)* in2 / 255 + in2_min)
				* K + O;
*)

(* revision History
hm 19.1.2007		rev 1.1
	changed outputs to real to avoid overflow of integer
	added offset for better cascading of scale functions
	changed from FB to function

hm	6. jan 2008		rev 1.2
	improved performance

hm	26. oct. 2008	rev 1.3
	code optimization

hm	3. nov. 2008	rev 1.4
	used wrong factor in formula

*)

END_FUNCTION

// POUs/Engineering/signal processing/SCALE_B4
FUNCTION SCALE_B4 : REAL
VAR_INPUT
	in1: BYTE;
	in2: BYTE;
	in3: BYTE;
	in4: BYTE;
	K : REAL;
	O : REAL;
END_VAR
VAR_INPUT CONSTANT
	in1_min: REAL;
	in1_max: REAL := 1000;
	in2_min: REAL;
	in2_max: REAL := 1000;
	in3_min: REAL;
	in3_max: REAL := 1000;
	in4_min: REAL;
	in4_max: REAL := 1000;
END_VAR

(*
version 1.4	3. nov. 2008
programmer 	hugo
tested by	tobias

	this functiob block can scale up to 4 inputs.
	the inputs have their min value at 0 and their max value at 255 while the min and max value can be either positive or negative.
	the inputs ramp between min and max values for the respective inputs to be between (0..255).
	the summed output is then scaled by an scale input K and a offset O can be added to the output.
	the min and max input configurations can be edited in the cfc editor by double clicking the symbol body.

*)

SCALE_B4 := 	(((in1_max - in1_min)* in1 + (in2_max - in2_min)* in2 + (in3_max - in3_min)* in3 + (in4_max - in4_min)* in4)* 0.003921569 + in1_min + in2_min + in3_min + in4_min) * K + O;


(* revision History
hm 19.1.2007		rev 1.1
	changed outputs to real to avoid overflow of integer
	added offset for better cascading of scale functions
	changed from fb to function

hm	6. jan 2008		rev 1.2
	improved performance

hm	26. oct. 2008	rev 1.3
	optimized code

hm	3. nov. 2008	rev 1.4
	used wrong factor in formula

*)

END_FUNCTION

// POUs/Engineering/signal processing/SCALE_B8
FUNCTION SCALE_B8 : REAL
VAR_INPUT
	in1: BYTE;
	in2: BYTE;
	in3: BYTE;
	in4: BYTE;
	in5: BYTE;
	in6: BYTE;
	in7: BYTE;
	in8: BYTE;
	K : REAL;
	O : REAL;
END_VAR
VAR_INPUT CONSTANT
	in1_min: REAL;
	in1_max: REAL := 1000;
	in2_min: REAL;
	in2_max: REAL := 1000;
	in3_min: REAL;
	in3_max: REAL := 1000;
	in4_min: REAL;
	in4_max: REAL := 1000;
	in5_min: REAL;
	in5_max: REAL := 1000;
	in6_min: REAL;
	in6_max: REAL := 1000;
	in7_min: REAL;
	in7_max: REAL := 1000;
	in8_min: REAL;
	in8_max: REAL := 1000;
END_VAR

(*
version 1.4	3. nov. 2008
programmer 	hugo
tested by	oscat

this functiob block can scale up to 8 inputs.
the inputs have their min value at 0 and their max value at 255 while the min and max value can be either positive or negative.
the inputs ramp between min and max values for the respective inputs to be between (0..255).
the summed output is then scaled by an scale input K and a offset O can be added to the output.
the min and max input configurations can be edited in the cfc editor by double clicking the symbol body.

*)

SCALE_B8 := 	(((in1_max - in1_min)* in1 + (in2_max - in2_min)* in2 + (in3_max - in3_min)* in3 + (in4_max - in4_min)* in4 +
				(in5_max - in5_min)* in5 + (in6_max - in6_min)* in6 + (in7_max - in7_min)* in7 + (in8_max - in8_min)* in8) * 0.003921569
				 + in1_min + in2_min + in3_min + in4_min + in5_min + in6_min + in7_min + in8_min) * K + O;


(* revision History
hm	19. jan.2007	rev 1.1
	changed outputs to real to avoid overflow of integer
	added offset for better cascading of scale functions

hm	6. jan. 2008	rev 1.2
	improved performance

hm	26. oct. 2008	rev 1.3
	code optimization

hm	3. nov. 2008	rev 1.4
	used wrong factor in formula

*)

END_FUNCTION

// POUs/Engineering/signal processing/SCALE_D
FUNCTION SCALE_D : REAL
VAR_INPUT
	X : DWORD;
	I_LO : DWORD;
	I_HI : DWORD;
	O_LO : REAL;
	O_HI : REAL;
END_VAR
VAR
END_VAR

(*
version 1.1	13. nov. 2008
programmer 	hugo
tested by	oscat

Scale_D is used to translate and scale a DWORD input x to a real output.
the input is limited to I_LO <= X <= I_HI.

*)

SCALE_D := (O_HI - O_LO) / DWORD_TO_REAL(I_HI - I_LO) * DWORD_TO_REAL(LIMIT(I_LO,X,I_HI) - I_LO) + O_LO;


(* revision history
hm	18. may. 2008	rev 1.0
	original version

hm	13. nov. 2008	rev 1.1
	corrected formula for negative gradient
*)

END_FUNCTION

// POUs/Engineering/signal processing/SCALE_R
FUNCTION SCALE_R : REAL
VAR_INPUT
	X : REAL;
	I_LO : REAL;
	I_HI : REAL;
	O_LO : REAL;
	O_HI : REAL;
END_VAR
VAR
END_VAR

(*
version 1.1	13. nov. 2008
programmer 	hugo
tested by	oscat

Scale_R is used to translate and scale a REAL input x to a real output.
the input is limited to I_LO <= X <= I_HI.

*)

SCALE_R := (O_HI - O_LO) / (I_HI - I_LO) * (LIMIT(I_LO,X,I_HI) - I_LO) + O_LO;


(* revision history
hm	18. may. 2008		rev 1.0
	original version

hm	13. nov. 2008	rev 1.1
	corrected formula for negative gradient

*)

END_FUNCTION

// POUs/Engineering/signal processing/SCALE_X2
FUNCTION SCALE_X2 : REAL
VAR_INPUT
	IN1: BOOL;
	IN2: BOOL;
	K : REAL;
	O : REAL;
END_VAR
VAR_INPUT CONSTANT
	IN1_MIN: REAL;
	IN1_MAX: REAL := 1000;
	IN2_MIN: REAL;
	IN2_MAX: REAL := 1000;
END_VAR

(*
version 1.1	26. oct. 2008
programmer 	hugo
tested by		tobias

	this functiob block can scale up to two inputs.
	the input can select between two values with true or false.
	the summed output is then scaled by an scale input K and a offset O can be added to the output.
	the min and max input configurations can be edited in the cfc editor by double clicking the symbol body.

*)

SCALE_X2 := (SEL(IN1,IN1_MIN, IN1_MAX)+ SEL(IN2,IN2_MIN, IN2_MAX))*k + o;


(* revision history
hm	19. jan, 2007	rev 1.0
	original version

hm	26. oct. 2008	rev 1.1
	code optimized

*)

END_FUNCTION

// POUs/Engineering/signal processing/SCALE_X4
FUNCTION SCALE_X4 : REAL
VAR_INPUT
	IN1: BOOL;
	IN2: BOOL;
	IN3: BOOL;
	IN4: BOOL;
	K : REAL;
	O : REAL;
END_VAR
VAR_INPUT CONSTANT
	IN1_MIN: REAL;
	IN1_MAX: REAL := 1000;
	IN2_MIN: REAL;
	IN2_MAX: REAL := 1000;
	IN3_MIN: REAL;
	IN3_MAX: REAL := 1000;
	IN4_MIN: REAL;
	IN4_MAX: REAL := 1000;
END_VAR

(*
version 1.1	26. oct. 2008
programmer 	hugo
tested by		tobias

	this function can scale up to 4 inputs.
	the input can select between two values with true or false.
	the summed output is then scaled by an scale input K and a offset O can be added to the output.
	the min and max input configurations can be edited in the cfc editor by double clicking the symbol body.

*)

SCALE_X4 := (SEL(IN1,IN1_MIN, IN1_MAX)+ SEL(IN2,IN2_MIN, IN2_MAX)+SEL(IN3,IN3_MIN, IN3_MAX)+ SEL(IN4,IN4_MIN, IN4_MAX))*k + o;


(* revision history
hm	19. jan. 2008	rev 1.0
	original version

hm	26. oct. 2008	rev 1.1
	optimized code
*)

END_FUNCTION

// POUs/Engineering/signal processing/SCALE_X8
FUNCTION SCALE_X8 : REAL
VAR_INPUT
	in1: BOOL;
	in2: BOOL;
	in3: BOOL;
	in4: BOOL;
	in5: BOOL;
	in6: BOOL;
	in7: BOOL;
	in8: BOOL;
	K : REAL;
	O : REAL;
END_VAR
VAR_INPUT CONSTANT
	in1_min: REAL;
	in1_max: REAL := 1000;
	in2_min: REAL;
	in2_max: REAL := 1000;
	in3_min: REAL;
	in3_max: REAL := 1000;
	in4_min: REAL;
	in4_max: REAL := 1000;
	in5_min: REAL;
	in5_max: REAL := 1000;
	in6_min: REAL;
	in6_max: REAL := 1000;
	in7_min: REAL;
	in7_max: REAL := 1000;
	in8_min: REAL;
	in8_max: REAL := 1000;
END_VAR

(*
version 1.2	24. jan. 2009
programmer 	hugo
tested by	oscat

this function can scale up to 4 inputs.
the input can select between two values with true or false.
the summed output is then scaled by an scale input K and a offset O can be added to the output.
the min and max input configurations can be edited in the cfc editor by double clicking the symbol body.

*)

SCALE_X8 := (SEL(IN1,IN1_MIN, IN1_MAX)+ SEL(IN2,IN2_MIN, IN2_MAX)+SEL(IN3,IN3_MIN, IN3_MAX)+ SEL(IN4,IN4_MIN, IN4_MAX)
				+SEL(IN5,IN5_MIN, IN5_MAX)+ SEL(IN6,IN6_MIN, IN6_MAX)+SEL(IN7,IN7_MIN, IN7_MAX)+ SEL(IN8,IN8_MIN, IN8_MAX))*k + o;



(* revision history
hm	19. jan. 2008	rev 1.0
	original version

hm	26. oct. 2008	rev 1.1
	optimized code

hm	24. jan. 2008	rev 1.2
	corrected error in formula
*)

END_FUNCTION

// POUs/Logic/generators/SCHEDULER
FUNCTION_BLOCK SCHEDULER
VAR_INPUT
	E0 : BOOL;
	E1 : BOOL;
	E2 : BOOL;
	E3 : BOOL;
END_VAR
VAR_INPUT CONSTANT
	T0, T1, T2, T3 : TIME;
END_VAR
VAR_OUTPUT
	Q0, Q1, Q2, Q3 : BOOL;
END_VAR
VAR
	init : BOOL;
	s0, s1, s2, s3 : TIME;
	tx : TIME;
	c : INT;
END_VAR


(*
version 1.0	28. sep 2008
programmer 	hugo
tested by		tobias

SCHEDULER is used to call programs or function blocks at specific intervals.
T0..T3 defines the interval times.

*)

(* read system_time *)
tx := DWORD_TO_TIME(T_PLC_MS());

IF NOT init THEN
	init := TRUE;
	s0 := tx - T0;
	s1 := tx - T1;
	s2 := tx - T2;
	s3 := tx - T3;
END_IF;

Q0 := Q1 := Q2 := Q3 :=FALSE;

CASE c OF
	0: 	IF tx - s0 >= T0 THEN
			Q0 := E0;
			s0 := tx;
		END_IF;
		c := 1;
	1: 	IF tx - s1 >= T1 THEN
			Q1 := E1;
			s1 := tx;
		END_IF;
		c := 2;
	2: 	IF tx - s2 >= T2 THEN
			Q2 := E2;
			s2 := tx;
		END_IF;
		c := 3;
	3: 	IF tx - s3 >= T3 THEN
			Q3 := E3;
			s3 := tx;
		END_IF;
		c := 0;
END_CASE;


(* revision history

hm 28. sep. 2008		rev 1.0
	original version


*)

END_FUNCTION_BLOCK

// POUs/Logic/generators/SCHEDULER_2
FUNCTION_BLOCK SCHEDULER_2
VAR_INPUT
	E0 : BOOL;
	E1 : BOOL;
	E2 : BOOL;
	E3 : BOOL;
END_VAR
VAR_INPUT CONSTANT
	C0, C1, C2, C3 : UINT;
	O0, O1, O2, O3 : UINT;
END_VAR
VAR_OUTPUT
	Q0, Q1, Q2, Q3 : BOOL;
END_VAR
VAR
	sx : UINT;
END_VAR


(*
version 1.0	29. sep 2008
programmer 	hugo
tested by		tobias

SCHEDULER_2 is used to call programs or function blocks at specific cycles.
C0..C3 defines after how many cycles the output becomes active.
O0..O3 defines a cycle offset at startup.

*)

Q0 := E0 AND (sx MOD C0 - O0 = 0);
Q1 := E1 AND (sx MOD C1 - O1 = 0);
Q2 := E2 AND (sx MOD C2 - O2 = 0);
Q3 := E3 AND (sx MOD C3 - O3 = 0);

(* increment cycle counter every cycle *)
sx := sx + 1;


(* revision history
hm 29. sep. 2008		rev 1.0
	original version


*)

END_FUNCTION_BLOCK

// POUs/Time&Date/SDT_TO_DATE
FUNCTION SDT_TO_DATE : DATE
VAR_INPUT
	DTI : SDT;
END_VAR
VAR
END_VAR


(*
version 1.0	18. oct 2008
programmer 	hugo
tested by	oscat

converts Structured date time (SDT) to Date Time

*)

SDT_TO_DATE := SET_DATE(DTI.YEAR, DTI.MONTH, DTI.DAY);



(* revision history

hm 18. oct. 2008	rev 1.0
	original version

*)

END_FUNCTION

// POUs/Time&Date/SDT_TO_DT
FUNCTION SDT_TO_DT : DT
VAR_INPUT
	DTI : SDT;
END_VAR
VAR
END_VAR


(*
version 1.0	18. oct 2008
programmer 	hugo
tested by	oscat

converts Structured date time (SDT) to Date Time

*)

SDT_TO_DT := SET_DT(DTI.YEAR, DTI.MONTH, DTI.DAY, DTI.HOUR, DTI.MINUTE, DTI.SECOND);



(* revision history

hm 18. oct. 2008	rev 1.0
	original version

*)

END_FUNCTION

// POUs/Time&Date/SDT_TO_TOD
FUNCTION SDT_TO_TOD : TOD
VAR_INPUT
	DTI : SDT;
END_VAR
VAR
END_VAR


(*
version 1.1	16. nov. 2008
programmer 	hugo
tested by	oscat

converts Structured date time (SDT) to Date Time

*)

SDT_TO_TOD := DWORD_TO_TOD(INT_TO_DWORD(DTI.HOUR) * 3600000 + INT_TO_DWORD(DTI.MINUTE) * 60000 + INT_TO_DWORD(DTI.SECOND) * 1000 + INT_TO_DWORD(DTI.MS));



(* revision history

hm 18. oct. 2008	rev 1.0
	original version

hm	16. nov. 2008	rev 1.1
	added typecasts to avoid warnings
*)

END_FUNCTION

// POUs/Time&Date/SECOND_OF_DT
FUNCTION SECOND_OF_DT : INT
VAR_INPUT
	XDT : DT;
END_VAR
VAR
END_VAR


(*
	version 1.0	6. jun. 2008
	programmer 	oscat
	tested BY	oscat

SECOND_OF_DT returns the current second (second of minute) of a DT variable

*)

SECOND_OF_DT := DWORD_TO_INT(DT_TO_DWORD(XDT) MOD 60);

(* revision history
hm		6.9.2008	rev 1.0
	original version

*)

END_FUNCTION

// POUs/Time&Date/SECOND_TO_TIME
FUNCTION SECOND_TO_TIME : TIME
VAR_INPUT
	IN : REAL;
END_VAR
VAR
END_VAR

(*
version 1.2	24. feb. 2009
programmer 	hugo
tested by		tobias

converts an amount of seconds in real to time
execution TIME on wago 750-841 =  17us 

*)

SECOND_TO_TIME := DWORD_TO_TIME(REAL_TO_DWORD(IN * 1000));

(* revision history
hm	4. aug. 2006	rev 1.0
	original version

hm	14. mar. 2008	rev 1.1
	rounded the input after the last digit

hm	24. feb. 2009	rev 1.2
	changed input to IN
*)

END_FUNCTION

// POUs/Engineering/signal processing/SEL2_OF_3
FUNCTION_BLOCK SEL2_OF_3
VAR_INPUT
	IN1 : REAL;
	IN2 : REAL;
	IN3 : REAL;
	D : REAL;
END_VAR
VAR_OUTPUT
	Y : REAL;
	W : INT;
	E : BOOL;
END_VAR
VAR
	D12: BOOL;
	D23: BOOL;
	D31: BOOL;
END_VAR

(*
	version 1.0	18. may. 2008
	programmer 	oscat
	tested BY		oscat

SEL2_OF_3 checks if 3 input Signals are within a distance D from each other and calculates the average of the 3 inputs do not offset more than D from each other.
If 1 input is more than D greater or smaller than any other input it will be ignored and the average will be calcualted from the remaining 2 Inputs.
In the case the Output is only calculated from 2 Inputs a Warning Output W will display the Number of the discarded Input. if none of the 3 Inputs are within the allowed Delata D from each other, 
an Error Output E is set True and the last valid Output will remain active until at least 2 Inputs are within a valid Range from each other.

*)

D12 := ABS(IN1-IN2) <= D;
D23 := ABS(IN2-IN3) <= D;
D31 := ABS(IN3-IN1) <= D;

IF (D12 AND D23) OR (D12 AND D31) OR (D23 AND D31) THEN
	(* all 3 inputs are valid *)
	Y := (IN1 + IN2 + IN3) / 3;
	E := FALSE;
	W := 0;
ELSIF D12 THEN
	(* only inut 1 and 2 are valid *)
	Y := (In1 + IN2) / 2;
	E := FALSE;
	W := 3;
ELSIF D23 THEN
	(* only inut 2 and 3 are valid *)
	Y := (In2 + IN3) / 2;
	E := FALSE;
	W := 1;
ELSIF D31 THEN
	(* only inut 3 and 1 are valid *)
	Y := (In3 + IN1) / 2;
	E := FALSE;
	W := 2;
ELSE
	(* no calculation possible *)
	E := TRUE;
	W := 4;
END_IF;


(* revision history
hm		18. may 2008	rev 1.0
	original version

*)

END_FUNCTION_BLOCK

// POUs/Engineering/signal processing/SEL2_OF_3B
FUNCTION_BLOCK SEL2_OF_3B
VAR_INPUT
	IN1 : BOOL;
	IN2 : BOOL;
	IN3 : BOOL;
	TD : TIME;
END_VAR
VAR_OUTPUT
	Q : BOOL;
	W : BOOL;
END_VAR
VAR
	TDEL : TON;
END_VAR

(*
	version 1.0	19. may. 2008
	programmer 	oscat
	tested BY		oscat

SEL2_OF_3B is used to connect 3 binary sensors to one signal. the output Q reflects the state of at least two inputs.
if two or more of the 3 inputs ate TRUE then Q will be TRUE and if two or more of the three inputs are FALSE then Q will be false.
the main putrpose is the connection of 3 redundant binary sensors.  
The output W will be active when one of the 3 inputs is of different state.
to avoid flickering while the sensors are switching the output W will become active after a programmed delay of TD.

*)

Q := (IN1 AND IN2) OR (IN1 AND IN3) OR (IN2 AND IN3);
TDEL(IN := (in1 XOR in2) OR (in1 XOR in3) OR (in2 XOR in3), PT := TD);
W := TDEL.Q;


(* revision history
hm		19. may 2008	rev 1.0
	original version

*)

END_FUNCTION_BLOCK

// POUs/Logic/FF edge triggered/SELECT_8
FUNCTION_BLOCK SELECT_8
VAR_INPUT
	E : BOOL;
	SET : BOOL;
	IN : BYTE;
	UP : BOOL;
	DN : BOOL;
	RST : BOOL;
END_VAR
VAR_OUTPUT
	Q0, Q1, Q2, Q3, Q4, Q5, Q6, Q7 : BOOL;
		STATE : INT;
END_VAR
VAR
	last_up: BOOL;
	last_dn : BOOL;
END_VAR

(*
	version 1.1	27. feb. 2009
	programmer 	hugo
	tested BY	tobias

select_8 selects one of 8 outputs at any time. the outputscan be selected by up or down keys and an independent anable switches all outouts off if set false


*)

IF rst THEN
	state := 0;
ELSIF set THEN
	state := IN;
ELSIF up AND NOT last_up THEN
	state := inc(state,1,7);
ELSIF dn AND NOT last_dn THEN
	state := inc(state,-1,7);
END_IF;
last_UP := UP;
last_DN := DN;

Q0 := FALSE;
Q1 := FALSE;
Q2 := FALSE;
Q3 := FALSE;
Q4 := FALSE;
Q5 := FALSE;
Q6 := FALSE;
Q7 := FALSE;

IF E THEN
	CASE state OF
		0: Q0 := TRUE;
		1: Q1 := TRUE;
		2: Q2 := TRUE;
		3: Q3 := TRUE;
		4: Q4 := TRUE;
		5: Q5 := TRUE;
		6: Q6 := TRUE;
		7: Q7 := TRUE;
	END_CASE;
END_IF;

(* revision history
hm	16. jan 2008	rev 1.0
	original version

hm	27. feb. 2009	rev 1.1
	renamed input en to e
*)

END_FUNCTION_BLOCK

// POUs/Engineering/sensor/SENSOR_INT
FUNCTION SENSOR_INT : REAL
VAR_INPUT
	Voltage : REAL;
	Current : REAL;
	RP : REAL;
	RS : REAL;
END_VAR
VAR
	RG: REAL;
END_VAR

(*
version 1.2	2 dec 2007
programmer 	hugo
tested by		tobias

this function calculates the real resistance of a sensor RX given a parasitic resistor in parallel to the sensor and an additional serial resistor.
for example a parasitic parallel resistor for a PT100 can be ignored but a series resistor is the cable to the sensor.
for a humidity sensor, the parallel resistor is more dramatic and needs to be considered.
the function allows to consider a parallel and serial resistor at the same time.
with this function and known parasitic serial and parallel resistors the true resistance of the sensor can be calculated.

*)

IF current <> 0 THEN
	RG := voltage / current;
	Sensor_Int := RP * ( RG - RS) / ( RP + RS - RG);
END_IF;

(* revisaion history

hm 20.1.2007	rev 1.1
	deleted input R0 which was not needed.

hm	2. dec 2007	rev 1.2
	corrected an error in formula and improoved speed
*)

END_FUNCTION

// POUs/Logic/generators/SEQUENCE_4
FUNCTION_BLOCK SEQUENCE_4
VAR_INPUT
	in0 : BOOL := TRUE;
	in1 : BOOL := TRUE;
	in2 : BOOL := TRUE;
	in3 : BOOL := TRUE;
	start : BOOL;
	rst : BOOL;
	wait0 : TIME;
	delay0 : TIME;
	wait1 : TIME;
	delay1 : TIME;
	wait2 : TIME;
	delay2 : TIME;
	wait3 : TIME;
	delay3 : TIME;
END_VAR
VAR_INPUT CONSTANT
	stop_on_error : BOOL;
END_VAR
VAR_OUTPUT
	Q0 : BOOL;
	Q1 : BOOL;
	Q2 : BOOL;
	Q3 : BOOL;
	CONVERSION_any : BOOL;
	run: BOOL;
	step : INT := -1;
	status : BYTE;
END_VAR
VAR
	last : TIME;
	edge : BOOL;
	tx: TIME;
	init: BOOL;
END_VAR

(*
version 1.4	17 sep 2007
programmer 	oscat
tested by	hans

sequence_4 enables run when a low to high transition is present on start.
a low to high transition on start will restart the sequencer at any time while a rst will hold the sequencer in reset while true.
after run is enabled with a rising edge on start the sequencer waits for wait0 on in0 to enable q0 which stays on for delay0.
the next cycle starts with wait1, continues with delay 1 and so on...
if an edge is not detected during the wait period, the sequencer will then display the error number on the status output.
the status numbers 1..4 are errors in step 0..3.
after the last step that sets q3, the sequencer leaves q3 on for delay3 and then resets to the initial state.
a step output will indicate the current step of the sequencer and will also be present with a fault condition.
after the first output is turened on the sequencer switches from q0 to q1 and so on, at any time there is only one output enabled.
if an input signal is not detected during a wait period, the sequencer will display the error number ( 1 for in0, 2 for in1 .... ).
when an error is present and the config variable stop_on_error is set then the sequencer will stop. otherwise it will continue.
The status output will also display 110 for waiting and 111 for sequence running.
*)

(* read sps timer *)
tx := DWORD_TO_TIME(T_PLC_MS());

(* initialize on startup *)
IF NOT init THEN
	last := tx;
	init := TRUE;
	status := 110;
END_IF;

(* asynchronous reset *)
IF rst THEN
	step := -1;
	Q0 := 0;
	Q1 := 0;
	Q2 := 0;
	Q3 := 0;
	status := 110;
	run := 0;

(* edge on start input restarts the sequencer *)
ELSIF start AND NOT edge THEN
	step := 0;
	last := tx;
	status := 111;
	Q0 := 0;
	Q1 := 0;
	Q2 := 0;
	Q3 := 0;
	run := 1;
END_IF;
edge := start;

(* check if stop on status is necessary *)
IF status > 0 AND status < 100 AND stop_on_error THEN RETURN; END_IF;

(* sequence is running *)
IF run AND step = 0 THEN
	IF NOT q0 AND in0 AND tx - last <= wait0 THEN
		Q0 := TRUE;
		last := tx;
	ELSIF NOT q0 AND tx - last > wait0 THEN
		status := 1;
		run := FALSE;
	ELSIF q0 AND tx - last >= delay0 THEN
		step := 1;
		last := tx;
	END_IF;
END_IF;
IF run AND step = 1 THEN
	IF NOT q1 AND in1 AND tx - last <= wait1 THEN
		Q0 := FALSE;
		Q1 := TRUE;
		last := tx;
	ELSIF NOT q1 AND Tx - last > wait1 THEN
		status := 2;
		q0 := FALSE;
		run := FALSE;
	ELSIF q1 AND tx - last >= delay1 THEN
		step := 2;
		last := tx;
	END_IF;
END_IF;
IF run AND step = 2 THEN
	IF NOT q2 AND in2 AND tx - last <= wait2 THEN
		Q1 := FALSE;
		Q2 := TRUE;
		last := tx;
	ELSIF NOT q2 AND Tx - last > wait2 THEN
		status := 3;
		q1 := FALSE;
		run := FALSE;
	ELSIF q2 AND tx - last >= delay2 THEN
		step := 3;
		last := tx;
	END_IF;
END_IF;
IF run AND step = 3 THEN
	IF NOT q3 AND in3 AND tx - last <= wait3 THEN
		Q2 := FALSE;
		Q3 := TRUE;
		last := tx;
	ELSIF NOT q3 AND Tx - last > wait3 THEN
		status := 4;
		q2 := FALSE;
		run := FALSE;
	ELSIF q3 AND tx - last >= delay3 THEN
		step := -1;
		q3 := FALSE;
		run := FALSE;
		status := 110;
	END_IF;
END_IF;
CONVERSION_any := q0 OR q1 OR q2 OR q3;

(*
hm 1.10.06		rev 1.1
	corrected delay logic to be after event and not before
	added any output

hm 1.12.06		rev 1.2
	corrected failure in sequence logic.
	added init at startup to prevent from initial error after start.

hm 17.1.2007		rev 1.3
	changed output fault to status for better compatibility with other modules (ESR).
	added stop on error functionality and setup variable
	default for inputs in0..3 is true.
	renamed variable state to step

hm	17.sep 2007		rev 1.4
	replaced time() with T_PLC_MS() for compatibility reasons

*)

END_FUNCTION_BLOCK

// POUs/Logic/generators/SEQUENCE_64
FUNCTION_BLOCK SEQUENCE_64
VAR_INPUT
	START : BOOL;
	SMAX : INT;
	PROG : ARRAY[0..63]OF TIME;
	RST : BOOL;
END_VAR
VAR_OUTPUT
	STATE : INT := -1;
	TRIG : BOOL;
END_VAR
VAR
	tx : TIME;
	edge: BOOL;
	last: TIME;
END_VAR


(*
version 1.0	29. jun. 2008
programmer 	hugo
tested by	oscat

sequence generates a sequence of states with a programmable length for each state.

*)

(* read system timer *)
tx := DWORD_TO_TIME(T_PLC_MS());
TRIG := FALSE;

IF RST THEN
	STATE := -1;

(* start sequence *)
ELSIF START AND NOT edge THEN
	STATE := 0;
	last := tx;
	TRIG := TRUE;

(* sequence generator *)
ELSIF (STATE >= 0) THEN
	IF (tx - last) >= PROG[STATE] THEN
		STATE := INC2(STATE, 1, -1, SMAX);
		last := tx;
		TRIG := TRUE;
	END_IF;
END_IF;

edge := START;



(* revision history
hm	29. jun. 2008
	original version

*)

END_FUNCTION_BLOCK

// POUs/Time&Date/SET_TOD
FUNCTION SET_TOD : TOD
VAR_INPUT
	hour : INT;
	minute : INT;
	second : REAL;
END_VAR
VAR
END_VAR

(*
version 1.5	16. mar 2008
programmer 	hugo
tested by	tobias

creates tod from hour minute and second 

*)

SET_TOD := DWORD_TO_TOD(REAL_TO_DWORD(SECOND * 1000) + INT_TO_DWORD(MINUTE) * 60000 + INT_TO_DWORD(HOUR) * 3600000);

(* revision history

hm		4.aug.2006		rev 1.0
	original version

hm		11. sep 2007	rev 1.1
	changed coding to avoid a compiler warning under twincat.

hm		1. nov 2007	rev 1.2
	changed coding to avoid possible overrun situation on möller ecp4

hm		2. Nov	2007	rev 1.3
	changed dword to DINT in calcualtion to avoid warnings with some compilers

hm		14. mar 2008	rev 1.4
	changed code to avoid rounding problem at last digit of millisecond

hm		16. mar. 2008	rev 1.5
	added type conversions to avoid warning under codesys 3.0
*)

END_FUNCTION

// POUs/Engineering/signal processing/SH
FUNCTION_BLOCK SH
VAR_INPUT
	in : REAL;
	CLK : BOOL;
END_VAR
VAR_OUTPUT
	out : REAL;
	trig : BOOL;
END_VAR
VAR
	edge : BOOL;
END_VAR

(*
version 1.1	16 jan 2007
programmer 	hugo
tested by		tobias

this sample and hold module samples an input at the rising edge of clk an stores it in out.
the out stays stable until the next rising clk edge appears.
a trigger output as active for one cycle when the output was updated.

*)

IF clk AND NOT edge THEN
	out := in;
	trig := TRUE;
ELSE;
	trig := FALSE;
END_IF;
edge := clk;

(* revision history

hm 16.1.2007	rev 1.1
	added trig output

*)

END_FUNCTION_BLOCK

// POUs/Engineering/signal processing/SH_1
FUNCTION_BLOCK SH_1
VAR_INPUT
	in : REAL;
	PT : TIME;
END_VAR
VAR_OUTPUT
	out : REAL;
	Trig : BOOL;
END_VAR
VAR
	last : TIME;
	tx: TIME;
END_VAR

(*
version 1.2	17 sep 2007
programmer 	hugo
tested by		tobias

this sample and hold module samples an input every PT seconds.
after a ample is taken the output Trig will be active for one cycle.

*)

(* read system time *)
tx := DWORD_TO_TIME(T_PLC_MS());

IF tx - last >= PT THEN
	last := tx;
	out := in;
	trig := TRUE;
ELSE
	trig := FALSE;
END_IF;

(* revision history

HM	6.1.2007	rev 1.1
	added trig output

HM	17.9.2007	rev 1.2
	replaced time() with T_PLC_MS() for compatibility reasons
*)

END_FUNCTION_BLOCK

// POUs/Engineering/signal processing/SH_2
FUNCTION_BLOCK SH_2
VAR_INPUT
	in : REAL;
	PT : TIME;
	N : INT := 16;
	disc : INT;
END_VAR
VAR_OUTPUT
	out : REAL;
	trig : BOOL;
	avg : REAL;
	high: REAL;
	low: REAL;
END_VAR
VAR
	M : INT;
	buf : ARRAY[0..15] OF REAL;
	buf2 : ARRAY[0..15] OF REAL;
	last : TIME;
	i : INT;
	start: INT;
	temp: REAL;
	stop: INT;
	tx: TIME;
	d2: INT;
END_VAR

(*
version 1.5	14. jun 2008
programmer 	hugo
tested by		tobias

this sample and hold module samples an input every PT seconds.
this sample and hold also does avg and other calculations with the input data.
an average is calculated over N samples while for this calculation disc samples are discarded,
disc = 0 all samples are averaged,
if disc = 1 the lowest value is ignored,
if disc = 2 the lowest and highest values are ignored, 
and so on.....

*)

(* read system time *)
tx := DWORD_TO_TIME(T_PLC_MS());
d2 := SHR(disc,1);

IF tx - last >= PT THEN
	last := tx;
	trig := TRUE;

	(* limit M to 0..16 *)
	M := LIMIT(1,N,16);

	(* edge detected lets take the sample *)
	FOR i := M - 1 TO 1 BY -1 DO buf2[i] := buf2[i-1]; END_FOR;
	buf2[0] := in;
	out := in;
	buf := buf2;

	(* sort the ARRAY lowest value AT 0 *)
	FOR start := 0 TO M - 2 DO
		FOR i := start+1 TO M - 1 DO
			IF buf[start] > buf[i] THEN
				temp := buf[start];
				buf[start] := buf[i];
				buf[i] := temp;
			END_IF;
		END_FOR;
	END_FOR;

	(* any calculation with the samples is here *)
	stop := M - 1 - d2;
	start := d2;
	IF NOT even(disc) THEN start := start + 1; END_IF;
	avg := 0;
	FOR i := start TO stop DO avg := avg + buf[i]; END_FOR;
	avg := avg / (stop - start +1);
	low := buf[start];
	high := buf[stop];
ELSE
	Trig := FALSE;
END_IF;

(* revision history
hm 20. jan. 2007	rev 1.1
	added input N to specify the amout of samples for average and high low calculations
	added trig output

hm 10. sep. 2007 	rev 1.2
	an error would be generated if N was set to 0, now n is forced to1 if set to 0.
	index was out of array.

hm	17. sep. 2007	rev 1.3
	replaced time() with t_plc_ms() for compatibility reasons

hm	6. jan. 2008	rev 1.4
	improved performance

hm	14. jun. 2008	rev 1.5
	set default for input N = 16
*)

END_FUNCTION_BLOCK

// POUs/Engineering/signal processing/SH_T
FUNCTION_BLOCK SH_T
VAR_INPUT
	IN : REAL;
	E : BOOL;
END_VAR
VAR_OUTPUT
	OUT : REAL;
END_VAR
VAR
END_VAR

(*
version 1.1	18. oct. 2008
programmer 	hugo
tested by	oscat

this sample and hold module samples an input while en is high.
during the high time of en the output follows in.
the out stays stable until the en goes high again.
*)

IF E THEN out := in; END_IF;



(* revision history
hm	1. sep. 2006	rev 1.0
	original version

hm	18. oct. 2008	rev 1.1
	changed input en to e for compatibility reasons

*)

END_FUNCTION_BLOCK

// POUs/Logic/gate logic/SHL1
FUNCTION SHL1 : DWORD
VAR_INPUT
	IN : DWORD;
	N : INT;
END_VAR
VAR CONSTANT
	temp : DWORD := 16#FFFF_FFFF;
END_VAR

(*
version 1.1	27 dec 2007
programmer 	hugo
tested by		tobias

SHL1 shifts N bits to the left filling the new bits with 1

*)

SHL1 := SHR(temp,32-N) OR SHL(IN,N);


(* revision history
hm	14.9.2007		rev 1.0
	original version

hm	27. dec 2007	rev 1.1
	changed code for better performance

*)

END_FUNCTION

// POUs/Logic/FF edge triggered/SHR_4E
FUNCTION_BLOCK SHR_4E
VAR_INPUT
	SET : BOOL;
	D0: BOOL;
	CLK: BOOL;
	RST: BOOL;
END_VAR
VAR_OUTPUT
	Q0: BOOL;
	Q1: BOOL;
	Q2: BOOL;
	Q3: BOOL;
END_VAR
VAR
	trig : R_TRIG;
END_VAR

(*
version 1.1	25. oct. 2008
programmer 	hugo
tested by		tobias

4 bit shift register with reset

*)

(* trig.Q signals a rising edge on clk *)
trig(clk := clk);

IF set OR rst THEN
	Q0 := Q1 := Q2 := Q3 := NOT RST;
ELSIF trig.Q THEN
	Q3 := Q2;
	Q2 := Q1;
	Q1 := Q0;
	Q0 := D0;
END_IF;



(* revision history
hm	4. aug. 2006	rev 1.0
	original version

hm	25. oct. 2008	rev 1.1
	optimized code

*)

END_FUNCTION_BLOCK

// POUs/Logic/FF edge triggered/SHR_4UDE
FUNCTION_BLOCK SHR_4UDE
VAR_INPUT
	SET : BOOL;
	D0: BOOL;
	D3: BOOL;
	CLK: BOOL;
	DN : BOOL;
	RST: BOOL;

END_VAR
VAR_OUTPUT
	Q0: BOOL;
	Q1: BOOL;
	Q2: BOOL;
	Q3: BOOL;
END_VAR
VAR
	trig : R_TRIG;
END_VAR

(*
version 1.1	25. oct. 2008
programmer 	hugo
tested by		tobias

4 bit shift register with reset up / down direction input

*)

(* trig.Q signals a rising edge on clk *)
trig(clk := clk);

IF set OR rst THEN
	Q0 := Q1 := Q2 := Q3 := NOT RST;
ELSIF trig.Q THEN
	IF dn THEN
		Q0 := Q1;
		Q1 := Q2;
		Q2 := Q3;
		Q3 := D3;
	ELSE
		Q3 := Q2;
		Q2 := Q1;
		Q1 := Q0;
		Q0 := D0;
	END_IF;
END_IF;



(* revision history
hm	4. aug. 2006	rev 1.0
	original version

hm	25. oct. 2008	rev 1.1
	optimized code

*)

END_FUNCTION_BLOCK

// POUs/Logic/FF edge triggered/SHR_8PLE
FUNCTION_BLOCK SHR_8PLE
VAR_INPUT
	Din : BOOL;
	Dload : BYTE;
	CLK: BOOL;
	UP: BOOL :=1;
	load : BOOL;
	RST: BOOL;
END_VAR
VAR_OUTPUT
	DOut: BOOL;
END_VAR
VAR
	edge : BOOL :=1;
	register : BYTE;
END_VAR

(*
version 1.0	4 aug 2006
programmer 	hugo
tested by	oscat

8 bit shift register with reset and parallel load
the register can shift up or down
it also has a serial input.
the Din input is on Bit0 for up shift and on bit 7 for down shift
the Dout output is on Bit7 for up shift and on bit 0 for down shift
paralle clock is performed clock synchron while a shift is performed first and then the register is reloaded


*)

(* flankenerkennung clk wird high und edge war high reset ist nicht aktiv und set ist nicht aktiv *)
IF CLK AND edge AND NOT rst THEN
	edge := FALSE;	(* flanke wurde erkannt und weitere flankenerkennung wird verhindert bis edge wieder true ist *)
	(* hier ist der code für das flankenevent *)
	IF UP THEN						(*shift up *)
		register := SHL(register,1);
		register.0 := Din;
		Dout := register.7;
	ELSE								(* shift down *);
		register := SHR(register,1);
		register.7 := Din;
		Dout := register.0;
	END_IF;
	IF load THEN							(* the byte on Din will be loaded if load = true *)
		register := Dload;
		IF up THEN Dout := register.7; ELSE Dout := register.0; END_IF;
	END_IF;
END_IF;
IF NOT clk THEN edge := TRUE; END_IF;	(* sobald clk wieder low wird warten auf nächste flanke *)
IF rst THEN									(* wenn reset aktiv dann ausgang rücksetzen *)
	register := 0;
	Dout := FALSE;
END_IF;

END_FUNCTION_BLOCK

// POUs/Logic/FF edge triggered/SHR_8UDE
FUNCTION_BLOCK SHR_8UDE
VAR_INPUT
	SET : BOOL;
	D0: BOOL;
	D7: BOOL;
	CLK: BOOL;
	DN : BOOL;
	RST: BOOL;
END_VAR
VAR_OUTPUT
	Q0: BOOL;
	Q1: BOOL;
	Q2: BOOL;
	Q3: BOOL;
	Q4: BOOL;
	Q5: BOOL;
	Q6: BOOL;
	Q7: BOOL;
END_VAR
VAR
	trig : R_TRIG;
END_VAR

(*
version 1.0	4 aug 2006
programmer 	hugo
tested by		tobias

8 bit shift register with reset

executioin TIME on wago 750-841 =  8 us
*)

(* trig.Q signals a rising edge on clk *)
trig(clk := clk);

IF set OR rst THEN
	Q0 := Q1 := Q2 := Q3 := Q4 := Q5 := Q6 := Q7 := NOT RST;
ELSIF trig.Q THEN
	IF dn THEN
		Q0 := Q1;
		Q1 := Q2;
		Q2 := Q3;
		Q3 := Q4;
		Q4 := Q5;
		Q5 := Q6;
		Q6 := Q7;
		Q7 := D7;
	ELSE
		Q7 := Q6;
		Q6 := Q5;
		Q5 := Q4;
		Q4 := Q3;
		Q3 := Q2;
		Q2 := Q1;
		Q1 := Q0;
		Q0 := D0;
	END_IF;
END_IF;



(* revision history
hm	4. aug. 2006	rev 1.0
	original version

hm	25. oct. 2008	rev 1.1
	optimized code

*)

END_FUNCTION_BLOCK

// POUs/Logic/gate logic/SHR1
FUNCTION SHR1 : DWORD
VAR_INPUT
	IN : DWORD;
	N : INT;
END_VAR
VAR CONSTANT
	temp : DWORD := 16#FFFF_FFFF;
END_VAR

(*
version 1.1	27 dec 2007
programmer 	hugo
tested by		tobias

SHR1 shifts N bits to the right filling the new bits with 1

*)

SHR1 := SHL(temp,32-N) OR SHR(IN,N);

(* revision history
hm	14.9.2007		rev 1.0
	original version

hm	27. dec 2007	rev 1.1
	changed code for better performance

*)

END_FUNCTION

// POUs/Mathematical/SIGMOID
FUNCTION SIGMOID : REAL
VAR_INPUT
	X : REAL;
END_VAR
VAR
END_VAR

(*
version 1.1	11.  mar 2008
programmer 	hugo
tested by	tobias

this function calculates the sigmoid function

*)

IF X > 20 THEN
	SIGMOID := 1;
ELSIF x < -85 THEN
	SIGMOID := 0;
ELSE
	SIGMOID := 1 / (1 + EXP(-X));
END_IF;

(* revision history
hm		10.12.2007		rev 1.0
	original version

hm		11. mar. 2008		rev 1.1
	extended range of valid inputs to +inv / -inv

*)

END_FUNCTION

// POUs/Mathematical/SIGN_I
FUNCTION SIGN_I : BOOL
VAR_INPUT
	IN : DINT;
END_VAR
VAR
END_VAR

(*
version 1.3	27. oct. 2008
programmer 	hugo
tested by	tobias

this function return true if the integer input is negative

*)

SIGN_I := in.31;

(* revision history
hm 3.3.2007	rev 1.1
	changed method of function for better compatibility to other systems

hm	1.12.2007	rev 1.2
	changed code to improve performance

hm	27. oct. 2008	rev 1.3
	changed type of input to dint
*)

END_FUNCTION

// POUs/Engineering/automation/SIGNAL_4
FUNCTION_BLOCK SIGNAL_4
VAR_INPUT
	IN1 : BOOL;
	IN2 : BOOL;
	IN3 : BOOL;
	IN4 : BOOL;
	TS : TIME;
END_VAR
VAR_INPUT CONSTANT
	S1 : BYTE := 2#1111_1111;
	S2 : BYTE := 2#1111_0000;
	S3 : BYTE := 2#1010_1010;
	S4 : BYTE := 2#1010_0000;
END_VAR
VAR_OUTPUT
	Q : BOOL;
END_VAR
VAR
	sig : SIGNAL;
END_VAR

(*
version 1.0	13 dec 2007
programmer 	hugo
tested by		tobias

this function generates one out of 4 signals specified by bit patterns S1 .. S4.
the selected pattern will be shifted with the step time TS.
In1 has higher priority then In2 which has higher priority then IN3 and in4 has the lowest priority.
ts defaults to 128 ms if not specified.
*)

(* an alarm is present read system time first *)
(* check if an alarm is present if yes set sig to the alarm pattern otherwise exit the routine *)
IF in1 THEN
	sig(in := TRUE, sig := s1, TS := TS);
ELSIF in2 THEN
	sig(in := TRUE, sig := s2, TS := TS);
ELSIF in3 THEN
	sig(in := TRUE, sig := s3, TS := TS);
ELSIF in4 THEN
	sig(in := TRUE, sig := s4, TS := TS);
ELSE
	sig(in := FALSE);
END_IF;

(* set the output *)
Q := sig.Q;


(* revision history
hm	13.12.2007		rev 1.0
	original version

*)

END_FUNCTION_BLOCK

// POUs/Mathematical/SINC
FUNCTION SINC : REAL
VAR_INPUT
	X : REAL;
END_VAR
VAR
END_VAR


(*
version 1.1	1. dec. 2008
programmer 	hugo
tested by	tobias

this function calculates the sinc function.

*)

IF X = 0 THEN
	SINC := 1;
ELSE
	SINC := SIN(x) / x;
END_IF;


(* revision histroy
hm	11. mar. 2008
	original version

hm	1.12.2007	rev 1.1
	changed code to improove performance

*)

END_FUNCTION

// POUs/Mathematical/Geometry/SPHERE_V
FUNCTION SPHERE_V : REAL
VAR_INPUT
	rx : REAL;
END_VAR
VAR
END_VAR

(*
version 1.2	22. feb 2008
programmer 	hugo
tested by		tobias

sphere_V calculates the Volume of a Sphere


*)

sphere_V := 4.188790205 * Rx * RX * RX;

(* revision histroy
hm	16. oct 2007	rev 1.0
	original version

hm	4. dec 2007		rev 1.1
	changed code for better performance

hm	22. feb 2008		rev 1.2
	changed code for better performance
*)

END_FUNCTION

// POUs/Engineering/automation/SRAMP
FUNCTION_BLOCK SRAMP
VAR_INPUT
	X : REAL;
	A_UP : REAL;
	A_DN :REAL;
	VU_MAX : REAL;
	VD_MAX : REAL;
	LIMIT_HIGH : REAL;
	LIMIT_LOW : REAL;
	RST : BOOL;
END_VAR
VAR_OUTPUT
	Y : REAL;
	V : REAL;
END_VAR
VAR
	cycle_time : TC_S;
	init: BOOL;
END_VAR


(*
	version 1.0	13 mar 2008
	programmer 	hugo
	tested by		tobias

RAMPS generates output signal which are slew rate and acceleration controlled.

*)

(* read the system_time in microseconds *)
cycle_time();

(* assure range of inputs *)
A_up := MAX(0,A_UP);
A_dn := MIN(0,A_dn);
VU_max := MAX(0,VU_max);
VD_max := MIN(0,VD_MAX);

(* calculate the output offset *)
IF rst OR NOT init THEN
	init := TRUE;
	Y := 0;
	V := 0;
ELSIF X = Y THEN
	v := 0;
ELSIF X > Y THEN
	(* output is too low >> ramp up and brake at the end *)
	(* accelerate the speed and limit to vu_max *)
	v := MIN(v + A_UP * cycle_time.TC, vu_max);
	(* calculate the max speed to be able to brake and select the lowest *)
	v := MIN(SQRT((Y-X) * 2 * A_DN), v);
	(* calculate the output and obey limits *)
	y := LIMIT(limit_low, y + MIN(v * cycle_time.TC, X-Y), limit_high);
ELSIF X < Y THEN
	(* output is too high >> ramp dn and brake at the end *)
	(* accelerate the speed and limit to vd_max *)
	v := MAX(v + A_DN * cycle_time.TC, vd_max);
	(* calculate the max speed to be able to brake and select the lowest *)
	v := MAX(-SQRT((Y-X) * 2 * A_UP), v);
	(* calculate the output and obey limits *)
	y := LIMIT(limit_low, y + MAX(v * cycle_time.TC, X-Y), limit_high);
END_IF;


(* revision history
hm		13. mar. 2008	rev 1.0
	original version

*)

END_FUNCTION_BLOCK

// POUs/Engineering/measurements/TC_S
FUNCTION_BLOCK TC_S
VAR_INPUT
END_VAR
VAR_OUTPUT
	TC : REAL;
END_VAR
VAR
	init: BOOL;
	tx: DWORD;
	last: DWORD;
END_VAR

(*
	version 1.1	16 mar 2008
	programmer 	hugo
	tested by		tobias

TC_S delivers the time it was last called on the output TC in seconds.

*)

(* read system timer *)
tx := T_PLC_US();

IF NOT init THEN
	init := TRUE;
	TC := 0;
ELSE
	tc := DWORD_TO_REAL(tx - last)*1.0E-6;
END_IF;
last := tx;

(* revision history
hm		13. mar. 2008	rev 1.0
	original version

hm		16. mar 2008	rev 1.1
	added type conversion to avoid warnings under codesys 3.0

*)

END_FUNCTION_BLOCK

// POUs/Logic/memory/STACK_16
FUNCTION_BLOCK STACK_16
VAR_INPUT
	Din : DWORD;
	RW : BOOL;
	E : BOOL;
	RST : BOOL;
END_VAR
VAR_OUTPUT
	Dout : DWORD;
	empty : BOOL := TRUE;
	full : BOOL;
END_VAR
VAR
	Stack : ARRAY[0..15] OF DWORD;
	N : INT := -1;
	top : INT := 15;
END_VAR

(*
version 1.3	27. oct. 2008
programmer 	hugo
tested by		oscat

16 Dword STACK memory

*)

IF rst THEN
	(* asynchronous reset for the fifo *)
	N := -1;
	Dout := 0;
	empty := TRUE;
	full := FALSE;
ELSIF E THEN
	IF RW AND NOT full THEN
		(* write action *)
		N := N + 1;
		full := N = TOP;
		empty := FALSE;
		stack[N] := Din;
	ELSIF NOT RW AND NOT empty THEN
		(* read from stack *)
		Dout := stack[N];
		N := N - 1;
		empty := N < 0;
		full := FALSE;
	END_IF;
END_IF;


(* revision history
hm	4. aug. 2006	rev 1.0
	original version

hm	19. feb 2008	rev 1.1
	performance improvements

hm	17. oct. 2008	rev 1.2
	deleted unnecessary init with 0

hm	27. oct. 2008	rev 1.3
	optimized performance
*)

END_FUNCTION_BLOCK

// POUs/Logic/memory/STACK_32
FUNCTION_BLOCK STACK_32
VAR_INPUT
	Din : DWORD;
	RW : BOOL;
	E : BOOL;
	RST : BOOL;
END_VAR
VAR_OUTPUT
	Dout : DWORD;
	empty : BOOL := TRUE;
	full : BOOL;
END_VAR
VAR
	Stack : ARRAY[0..31] OF DWORD;
	N : INT := -1;
	top : INT := 31;
END_VAR

(*
version 1.3	27. oct. 2008
programmer 	hugo
tested by		oscat

32 Dword STACK memory
*)

IF rst THEN
	(* asynchronous reset for the fifo *)
	N := -1;
	Dout := 0;
	empty := TRUE;
	full := FALSE;
ELSIF E THEN
	IF RW AND NOT full THEN
		(* write action *)
		N := N + 1;
		full := N = TOP;
		empty := FALSE;
		stack[N] := Din;
	ELSIF NOT RW AND NOT empty THEN
		(* read from stack *)
		Dout := stack[N];
		N := N - 1;
		empty := N < 0;
		full := FALSE;
	END_IF;
END_IF;


(* revision history
hm	4. aug. 2006	rev 1.0
	original version

hm	19. feb 2008	rev 1.1
	performance improvements

hm	17. oct. 2008	rev 1.2
	deleted unnecessary init with 0

ks	27. oct. 2008	rev 1.3
	optimized performance
*)

END_FUNCTION_BLOCK

// POUs/Engineering/signal processing/STAIR
FUNCTION STAIR : REAL
VAR_INPUT
	X : REAL;
	D : REAL;
END_VAR
VAR
END_VAR


(*
version 1.3	26. oct. 2008
programmer 	oscat
tested by		tobias

the function stair converts an anlog input signal to a staircase like output.
D is the step width for the output signal.
if D = 0 then the output follows the input without a chage.
*)

IF D > 0 THEN
	STAIR := DINT_TO_REAL(REAL_TO_DINT(X / D)) * D;
ELSE
	STAIR := X;
END_IF;


(* code for rev 1.2
temp := MODR(X, D);
IF ABS(temp) < D * 0.5 THEN
	stair := X - temp;
ELSE
	IF X > 0 THEN stair := X - temp + D; ELSE stair := X - temp - D; END_IF;
END_IF;
*)


(* revision history
hm	28 jan 2007		rev 1.0
	original version

hm	27 dec 2007		rev 1.1
	changed code for better performance

hm	6. jan 2008		rev 1.2
	further performance improvement

hm	26. oct. 2008		rev 1.3
	optimized code
*)

END_FUNCTION

// POUs/Engineering/signal processing/STAIR2
FUNCTION_BLOCK STAIR2
VAR_INPUT
	X : REAL;
	D : REAL;
END_VAR
VAR_OUTPUT
	Y: REAL;
END_VAR
VAR
END_VAR


(*
version 1.3	26. oct. 2008
programmer 	hugo
tested by		oscat

the function stair2 converts an anlog input signal to a staircase like output.
D is the step width for the output signal. the output will use D as a hysteresis for a stairchange.
if D = 0 then the output follows the input without a chage.
*)

IF D > 0 THEN
	IF X >= Y + D OR X <= Y - D THEN Y := FLOOR(X/D) * D; END_IF;
ELSE
	Y := X;
END_IF;


(* code for rev 1.2
IF X >= Y AND X >= 0 THEN
	Y := DINT_TO_REAL(TRUNC(X / D)) * D;
ELSIF X < Y AND X >= 0 THEN
	Y := DINT_TO_REAL(TRUNC(X/d) + 1) * D;
ELSIF X >= Y AND X < 0 THEN
	Y := DINT_TO_REAL(TRUNC(X/D)-1) * D;
ELSIF X < Y AND X < 0 THEN
	Y := DINT_TO_REAL(TRUNC(X/D)) *D;
END_IF;
*)

(* revision history
hm	28 jan 2007		rev 1.0
	original version

hm	27. dec 2007	rev 1.1
	changed code for better performance

hm	30. jun. 2008	rev 1.2
	added type conversions to avoid warnings under codesys 3.0																																																																																																																																																																																																																																																											

ks	26. oct. 2008	rev 1.3
	improved code
*)

END_FUNCTION_BLOCK

// POUs/Logic/FF pulse triggered/STORE_8
FUNCTION_BLOCK STORE_8
VAR_INPUT
	Set : BOOL;
	D0,D1, D2, D3, D4, D5, D6, D7 : BOOL;
	Clr : BOOL;
	Rst : BOOL;
END_VAR
VAR_OUTPUT
	Q0, Q1, Q2, Q3, Q4, Q5, Q6, Q7 : BOOL;
END_VAR
VAR
	edge: BOOL;
END_VAR

(*
version 1.1	30. oct. 2008
programmer 	hugo
tested by	oscat

Store_4 stores up to 4 boolean inputs until a reset is clearing the outputs.
the respective output is set with a true at the respective input and stays true until a reset is generated.
a set input is used to set all outputs true at the same time, independent of their inputs.
a clear input is used to reset only the lowest priority of the outputs one at a time.
the lowest priority is q3.

*)

IF rst OR set THEN
	q0 := q1 := q2 := q3 := q4 := q5 := q6 := q7 := NOT rst;
ELSE
	IF D0 THEN Q0 := TRUE; END_IF;
	IF D1 THEN Q1 := TRUE; END_IF;
	IF D2 THEN Q2 := TRUE; END_IF;
	IF D3 THEN Q3 := TRUE; END_IF;
	IF D4 THEN Q4 := TRUE; END_IF;
	IF D5 THEN Q5 := TRUE; END_IF;
	IF D6 THEN Q6 := TRUE; END_IF;
	IF D7 THEN Q7 := TRUE; END_IF;

	IF clr AND NOT edge THEN
		IF q0 THEN q0 := FALSE;
		ELSIF q1 THEN q1 := FALSE;
		ELSIF q2 THEN q2 := FALSE;
		ELSIF q3 THEN q3 := FALSE;
		ELSIF q4 THEN q4 := FALSE;
		ELSIF q5 THEN q5 := FALSE;
		ELSIF q6 THEN q6 := FALSE;
		ELSE q7 := FALSE;
		END_IF;
	END_IF;
	edge := clr;
END_IF;


(* revision history
hm	25.12.2007	rev 1.0
	original version

hm	30. oct. 2008	rev 1.1
	optimized performance
*)

END_FUNCTION_BLOCK

// POUs/Network/STRING_TO_URL
FUNCTION STRING_TO_URL : URL
VAR_INPUT
	STR : STRING(255);
	DEFAULT_PROTOCOL : STRING(20);
	DEFAULT_PATH : STRING(80);
END_VAR
VAR
	pos: INT;
	pos2: INT;
END_VAR

(*
version 1.0	18. apr. 2008
programmer 	hugo
tested by		oscat

URL splits a unifrom resource locator in its conponents.

*)

(*

http://hans:geheim@www.example.org:80/demo/example.cgi?land=de&stadt=aa#abschnitt1
|         |         |                  |                                |   |                                    |                                    |
|         |         |                 Host                         |   Pfad                            Query                           Anker
|         |         Passwort                                  Port
|        Benutzer
Protokoll

*)

(* check if string is empty and return empty url *)
IF STR = '' THEN RETURN; END_IF;

(* extract the protocol *)
(* first we check if the optional protocol is specified ending with a :// *)
pos := FIND(STR, '://');
IF pos > 0 THEN
	(* store protocol and restore the rest of url in temp *)
	STRING_TO_URL.PROTOCOL := LEFT(STR, pos - 1);
	STRING_TO_URL.DOMAIN := RIGHT(STR, LEN(STR) - pos - 2);
ELSE
	STRING_TO_URL.DOMAIN := STR;
	STRING_TO_URL.PROTOCOL := DEFAULT_PROTOCOL;
END_IF;

(* extract user and password if present ending with a @ *)
pos := FIND(STRING_TO_URL.DOMAIN, '@');
IF pos > 0 THEN
	(* extract user *)
	pos2 := FIND(STRING_TO_URL.DOMAIN,':')+1;
	IF pos2 > 1 AND pos2 <= pos THEN
		STRING_TO_URL.USER := LEFT(STRING_TO_URL.DOMAIN,pos2 - 2);
		STRING_TO_URL.PASSWORD := MID(STRING_TO_URL.DOMAIN, pos - pos2, pos2);
	ELSE
		STRING_TO_URL.USER := LEFT(STRING_TO_URL.DOMAIN, pos - 2);
		STRING_TO_URL.PASSWORD := '';
	END_IF;
	STRING_TO_URL.DOMAIN := RIGHT(STRING_TO_URL.DOMAIN, LEN(STRING_TO_URL.DOMAIN) - pos);
ELSE
	STRING_TO_URL.USER := '';
	STRING_TO_URL.PASSWORD := '';
END_IF;

(* extract anchor *)
pos := FIND(STRING_TO_URL.DOMAIN, '#');
IF pos > 0 THEN
	STRING_TO_URL.ANCHOR := RIGHT(STRING_TO_URL.DOMAIN, LEN(STRING_TO_URL.DOMAIN) - pos);
	STRING_TO_URL.DOMAIN := LEFT(STRING_TO_URL.DOMAIN, pos - 1);
ELSE
	STRING_TO_URL.ANCHOR := '';
END_IF;

(* extract query  *)
pos := FIND(STRING_TO_URL.DOMAIN, '?');
IF pos > 0 THEN
	STRING_TO_URL.QUERY := RIGHT(STRING_TO_URL.DOMAIN, LEN(STRING_TO_URL.DOMAIN) - pos);
	STRING_TO_URL.DOMAIN := LEFT(STRING_TO_URL.DOMAIN, pos - 1);
ELSE
	STRING_TO_URL.QUERY := '';
END_IF;

(* extract path  *)
pos := FIND(STRING_TO_URL.DOMAIN, '/');
IF pos > 0 THEN
	STRING_TO_URL.PATH := RIGHT(STRING_TO_URL.DOMAIN, LEN(STRING_TO_URL.DOMAIN) - pos + 1);
	STRING_TO_URL.DOMAIN := LEFT(STRING_TO_URL.DOMAIN, pos - 1);
ELSE
	STRING_TO_URL.PATH := DEFAULT_PATH;
END_IF;

(* extract port and leave domain *)
pos := FIND(STRING_TO_URL.DOMAIN, ':');
IF pos > 0 THEN
	STRING_TO_URL.PORT := STRING_TO_WORD(RIGHT(STRING_TO_URL.DOMAIN, LEN(STRING_TO_URL.DOMAIN) - pos));
	STRING_TO_URL.DOMAIN := LEFT(STRING_TO_URL.DOMAIN, pos - 1);
ELSE
	STRING_TO_URL.PORT := 0;
END_IF;




(* revision history
hm		18. apr 2008	rev 1.0
	original version

*)

END_FUNCTION

// POUs/Logic/gate logic/SWAP_BYTE
FUNCTION SWAP_BYTE : WORD
VAR_INPUT
	IN : WORD;
END_VAR
VAR
END_VAR

(*
version 1.0	4 feb 2008
programmer 	hugo
tested by		tobias

This function swaps the high and low byte of the word in.

*)

SWAP_BYTE := ROL(in,8);


(* revision history
hm		4. feb 2008	rev 1.0
	original version

*)

END_FUNCTION

// POUs/Logic/gate logic/SWAP_BYTE2
FUNCTION SWAP_BYTE2 : DWORD
VAR_INPUT
	IN : DWORD;
END_VAR
VAR
END_VAR

(*
version 1.0	4 feb 2008
programmer 	hugo
tested by		tobias

This function reverses the byte order in the dword.

*)

Swap_Byte2 := (ROR(in,8) AND 16#FF00FF00) OR (ROL(in,8) AND 16#00FF00FF);

(* revision history
hm		4. feb 2008	rev 1.0
	original version

*)

END_FUNCTION

// POUs/Building/electrical/SWITCH_I
FUNCTION_BLOCK SWITCH_I
VAR_INPUT
	set : BOOL;
	in : BOOL;
	rst : BOOL;
END_VAR
VAR_INPUT CONSTANT
	T_debounce : TIME := T#10ms;
	T_reconfig : TIME := T#1s;
	T_on_max : TIME := T#0h;
END_VAR
VAR_OUTPUT
	Q : BOOL;
END_VAR
VAR
	state : BYTE;
	edge : BOOL;
	r_edge : BOOL;
	T_on : TIME;
	tx: TIME;
END_VAR

(*
version 1.1	15 sep 2007
programmer 	oscat
tested by	oscat

this is an intelligent switch interface which has an autodetect feature for in and it will detect the type of switch connected automatically
the input can be connected to low active pulses, high active pulses and on/off switch.
it will automatically adjust to the correct type without manual adjustment
a configurable debounce timer will debounce input signals
if t_on_max is set to anything other then 0 the output will be turned off after the max on time is reached.

*)

(* read system time *)
tx := DWORD_TO_TIME(T_PLC_MS());

(* asynchronous set and reset first *)
IF set AND NOT rst THEN
	Q := TRUE;
	T_on := tx;
ELSIF rst THEN
	Q := FALSE;
(* check FOR input edge AND start debounce timer *)
ELSIF (in XOR edge) AND NOT (state = 1) THEN
	state := 1;
	T_on := Tx;
(* edge was detected and debounce time elapsed *)
ELSIF (state = 1) AND (Tx - t_debounce >= T_on) THEN
	state := 2;
	(* react on rising or falling edge depending on r_edge *)
	IF r_edge XOR in THEN Q := NOT Q; END_IF;
(* wait for T_reconfig and adjust r_edge *)
ELSIF state = 2 AND Tx - t_reconfig >= T_on THEN
	r_edge := in;
END_IF;
IF Q AND T_on_max > t#0ms AND Tx >= T_on + T_on_max THEN
	Q := FALSE;
END_IF;
edge := in;

(* revision history

hm	4 aug 2006	rev 1.0
	original version

hm	15.9.2007	rev 1.1
	replaced Time() with T_PLC_MS for compatibility and performance reasons

*)

END_FUNCTION_BLOCK

// POUs/Building/electrical/SWITCH_X
FUNCTION_BLOCK SWITCH_X
VAR_INPUT
	IN1 : BOOL;
	IN2 : BOOL;
	IN3 : BOOL;
	IN4 : BOOL;
	IN5 : BOOL;
	IN6 : BOOL;
END_VAR
VAR_OUTPUT
	Q1 : BOOL;
	Q2 : BOOL;
	Q3 : BOOL;
	Q4 : BOOL;
	Q5 : BOOL;
	Q6 : BOOL;
	Q31 : BOOL;
	Q41 : BOOL;
	Q51 : BOOL;
	Q61 : BOOL;
	Q32 : BOOL;
	Q42 : BOOL;
	Q52 : BOOL;
	Q62 : BOOL;
END_VAR
VAR_INPUT CONSTANT
	t_debounce : TIME := t#50ms;
END_VAR
VAR
	init : BOOL;
	T1, T2, T3, T4, T5, T6 : TOF;
	tx: TIME;
	x1: BOOL;
	x2: BOOL;
	E1, E2 : BOOL;
END_VAR

(*
version 1.0	15 Feb 2007
programmer 	oscat
tested by	oscat

*)

(* initialize on startup *)
IF NOT init THEN
	init := TRUE;
	IF t_debounce < t#50ms THEN tx := t#50ms; ELSE tx := t_debounce; END_IF;
	T1(PT := Tx);
	T2(PT := Tx);
	T3(PT := Tx);
	T4(PT := Tx);
	T5(PT := Tx);
	T6(PT := Tx);
ELSE
	Q1 := FALSE;
	Q2 := FALSE;
	Q3 := FALSE;
	Q4 := FALSE;
	Q5 := FALSE;
	Q6 := FALSE;
	Q31 := FALSE;
	Q41 := FALSE;
	Q51 := FALSE;
	Q61 := FALSE;
	Q32 := FALSE;
	Q42 := FALSE;
	Q52 := FALSE;
	Q62 := FALSE;
END_IF;

(* read inputs and debounce *)
	T1(IN := IN1);
	T2(IN := IN2);
	T3(IN := IN3);
	T4(IN := IN4);
	T5(IN := IN5);
	T6(IN := IN6);

(* detect edge of IN1 and IN2 *)
IF t1.Q AND NOT E1 THEN X1 := TRUE; END_IF;
IF t2.Q AND NOT E2 THEN X2 := TRUE; END_IF;

IF t1.Q THEN
	IF t3.q THEN
		q31 := TRUE;
		X1 := FALSE;
	ELSIF t4.q THEN
		q41 := TRUE;
		X1 := FALSE;
	ELSIF t5.q THEN
		q51 := TRUE;
		X1 := FALSE;
	ELSIF t6.q THEN
		q61 := TRUE;
		X1 := FALSE;
	END_IF;
ELSIF t2.Q THEN
	IF t3.q THEN
		q32 := TRUE;
		X2 := FALSE;
	ELSIF t4.q THEN
		q42 := TRUE;
		X2 := FALSE;
	ELSIF t5.q THEN
		q52 := TRUE;
		X2 := FALSE;
	ELSIF t6.q THEN
		q62 := TRUE;
		X2 := FALSE;
	END_IF;
(* in1 was active alone *)
ELSIF NOT T1.Q AND E1 AND X1 THEN
	Q1 := TRUE;
	X1 := FALSE;
ELSIF NOT T2.Q AND E2 AND X2 THEN
	Q2 := TRUE;
	X2 := FALSE;
ELSIF T3.Q THEN
	Q3 := TRUE;
ELSIF T4.Q THEN
	Q4 := TRUE;
ELSIF T5.Q THEN
	Q5 := TRUE;
ELSIF T6.Q THEN
	Q6 := TRUE;
END_IF;

(* save state of in1 and in2 *)
E1 := T1.Q;
E2 := T2.Q;

END_FUNCTION_BLOCK

// POUs/Building/HLK/T_AVG24
FUNCTION_BLOCK T_AVG24
VAR_INPUT
	TS : INT;
	DTI : DT;
	RST : BOOL;
END_VAR
VAR_INPUT CONSTANT
	T_FILTER : TIME := T#10m;
	SCALE : REAL := 1.0;
	OFS : REAL;
END_VAR
VAR_OUTPUT
	TA : REAL;
	TP : BOOL;
END_VAR
VAR_IN_OUT
	T24 : REAL;
	T24_MAX : REAL;
	T24_MIN : REAL;
END_VAR
VAR
	samples : ARRAY[0..47] OF INT;
	pos : INT;
	init: BOOL;
	ft1 : FILTER_I;
	sum : DINT;
	last: DT;
END_VAR
VAR
	tmp_max : INT;
	tmp_min : INT;
	i: INT;
END_VAR

(*
version 1.0	8. feb. 2009
programmer 	hugo
tested by	oscat

this function calculates the averaged daytime temperature by taking 48 samples over one day.
a trigger tp will be true for one cycle when the output is updated.
using the input scale the outputs can be adjusted to different scales.

*)

(* first filter the sensor readings *)
ft1(X := TS, T := T_FILTER);

IF rst OR NOT init THEN
	init := TRUE;
	IF T24 = -1000 THEN t24 := INT_TO_REAL(ft1.Y) / 10.0; END_IF;
	FOR pos := 0 TO 47 DO
		samples[pos] := REAL_TO_INT(T24 * 10.0);
	END_FOR;
	pos := 0;
	sum := INT_TO_DINT(samples[0]) * 48;
	(* calculate the output value *)
	TA := (INT_TO_REAL(ft1.Y)/10.0 + OFS) * SCALE;
	T24 := (DINT_TO_REAL(sum) / 480.0 + OFS) * SCALE;
	tp := TRUE;
ELSIF DT_TO_DWORD(dti) / 60 MOD 30 = 0 AND DTI > last THEN
	(* make sure we onlyexecute once every 30 mins *)
	last := DTI + T#1m;
	(* sample the temperature every 30 mins and store in ring buffer samples *)
	(* sum always holds the sum of the array *)
	(* subtract the oldest sample from sum *)
	sum := sum - INT_TO_DINT(samples[pos]);
	(* strore the new sample *)
	samples[pos] := ft1.Y;
	(* add the new sample to sum *)
	sum := sum + INT_TO_DINT(samples[pos]);
	(* increment the counter for the next sample *)
	pos := INC1(pos, 48);
	(* calculate the output value *)
	TA := (INT_TO_REAL(ft1.Y)/10.0 + OFS) * SCALE;
	T24 := (DINT_TO_REAL(sum) / 480.0 + OFS) * SCALE;
	(* calculate the min and max over the last 24 hours *)
	tmp_max := -32000;
	tmp_min := 32000;
	FOR i := 0 TO 47 DO
		tmp_max := MAX(tmp_max, samples[i]);
		tmp_min := MIN(tmp_min, samples[i]);
	END_FOR;
	T24_MAX := (INT_TO_REAL(tmp_max) / 10.0 + OFS) * SCALE;
	T24_MIN := (INT_TO_REAL(tmp_min) / 10.0 + OFS) * SCALE;
	tp := TRUE;
ELSE
	tp := FALSE;
END_IF;





(* revision history
hm	3. nov. 2008	rev 1.0
	original version

hm	8. feb. 2009	rev 1.1
	changes sign of OFS
	added outputs t24_min and t24_max

*)

END_FUNCTION_BLOCK

// POUs/Mathematical/TANC
FUNCTION TANC : REAL
VAR_INPUT
	X : REAL;
END_VAR
VAR
END_VAR


(*
version 1.0	23. oct. 2008
programmer 	hugo
tested by	oscat

this function calculates the tanc function.

*)

IF X = 0 THEN
	TANC := 1;
ELSE
	TANC := TAN(x) / x;
END_IF;


(* revision histroy
hm	23. oct. 2008
	original version


*)

END_FUNCTION

// POUs/Mathematical/TANH
FUNCTION TANH : REAL
VAR_INPUT
	X : REAL;
END_VAR
VAR
END_VAR


(*
version 1.2	10. mar 2008
programmer 	hugo
tested by	tobias

this function calculates the tangens hyperbolicus

*)

IF X > 20 THEN
	tanH := 1;
ELSIF X < -20 THEN
	tanH := -1;
ELSE
	tanH := 1 - 2 / (EXP(2 * x) + 1);
END_IF;

(* revision hisdtory
hm		12.1.2007		rev 1.0
	original version

hm		1.12.2007		rev 1.1
	changed code to improve performance

hm		10. mar 2008	rev 1.2
	corrected an error in formula
	extended range of valid inputs to +/- INV
*)

END_FUNCTION

// POUs/Engineering/automation/TANK_LEVEL
FUNCTION_BLOCK TANK_LEVEL
VAR_INPUT
	LEVEL : BOOL;
	LEAK : BOOL;
	ACLR : BOOL;
END_VAR
VAR_INPUT CONSTANT
	MAX_VALVE_TIME : TIME;
	LEVEL_DELAY_TIME : TIME;
END_VAR
VAR_OUTPUT
	VALVE : BOOL;
	ALARM : BOOL;
	STATUS : BYTE;
END_VAR
VAR
	cx : ACTUATOR_COIL;
	tn : TON;
	tl : TONOF;
	open: BOOL;
END_VAR


(*
version 1.0	27 feb 2007
programmer 	hugo
tested by		tobias

*)

(* preprocess the level information *)
tl(in := level, T1 := level_delay_time, T2 := level_delay_time);
open := tl.Q;

(* start logic *)
IF ALARM THEN
	(* check for ACLR if ALARM is present *)
	IF ACLR THEN
		ALARM := FALSE;
		STATUS := 101; (* aclr pressed *)
		cx(in := FALSE);
	END_IF;
	RETURN;
ELSIF LEAK THEN
	(* leakeage detected *)
	cx(in := FALSE);
	ALARM := TRUE;
	STATUS := 1;	(* leakeage error *)
ELSIF open THEN
	(* valve needs to be opened because level is too low *)
	cx(in := TRUE);
	STATUS := 102; (* valve open by low level *)
ELSE
	(* valve needs to be closed *)
	cx(in := FALSE);
	STATUS := 100; (* valve idle *)
END_IF;

(* check if valve is open too long and generate alarm if necessary *)
tn(in := cx.out AND (MAX_VALVE_TIME > T#0s), PT := MAX_VALVE_TIME);
IF tn.Q THEN
	ALARM := TRUE;
	STATUS := 2; (* overtime error *)
	cx(in := FALSE);
END_IF;

(* set output signal *)
VALVE := cx.out;

END_FUNCTION_BLOCK

